//GENERAL
OP40_Auto:					BOOL;
OP40_HomeRunning:			BOOL;
OP40_ErrorActive:			BOOL;
OP40_Home_PB:				BOOL;
OP40_Work_PB:				BOOL;
OP40_ManualSafetyBypass:	BOOL;
OP40_LightCurtainBypass:	BOOL;
OP40_OperationCompleted:	BOOL;
OP40_LampCheck:				BOOL;
OP40_MachineLamp:			BOOL;
OP40_ComponentOk:			BOOL;
OP40_ComponentNok:			BOOL;
OP40_RepeatBit:				BOOL;
OP40_HomingResetBit:		BOOL;
OP40_ControlledByRobo:		BOOL;
OP40_Any_Bypass:			BOOL;
OP40_ManualModeStatus:		INT;
OP40_ManualModeWord:		INT;
OP40_AutoRunning:			BOOL;
OP40_StepRunning:			BOOL;
OP40_StartEnable:   		BOOL;
OP40_Machine_Stop: 			BOOL;
OP40_AutoSeq:				INT;
OP40_LH_AutoSeq: 			INT;
OP40_RH_AutoSeq: 			INT;
OP40_Homing_Seq:			INT;
OP40_HomeConditionOK:   	BOOL;
OP40_Safety_OK:				BOOL;
OP40_Mode_Ack:				BOOL;
OP40_Temp_hmeOK:			BOOL;
OP40_Stop_Request: BOOL;

//Automatic_Run:				BOOL;

OP40_Prev_Stat_Operation_Completed: BOOL;
OP40_Prev_Comp_Status: INT;
OP40_Prev_LH_COMP_OK:BOOL;
OP40_Prev_LH_COMP_NOK:BOOL;
OP40_Prev_RH_COMP_OK:BOOL;
OP40_Prev_RH_COMP_NOK:BOOL;
OP40_LH_Operation_Completed:BOOL;
OP40_RH_Operation_Completed:BOOL;

//ModeSelection Outputs
//OP130_AutoSelected:		    BOOL;
OP40_ManualSelected:		BOOL;
OP40_StepSelected:			BOOL;
OP40_AutoSelected:		    BOOL;


//HMI Tags(From HMI)
OP40_HMI_AutoMode:						BOOL;
OP40_HMI_ManualMOde:					BOOL;
OP40_HMI_StepMode:						BOOL;
OP40_HMI_CycleStart:					BOOL;
OP40_HMI_Cycle_Start:					BOOL;
OP40_HMI_Reset:						    BOOL;
OP40_HMI_Homing:						BOOL;
SR40_Vert_Servo_Max_Lim:				BOOL;



//Servo
SR40_Vert_servo : FB_Axis;
SR40_Vert_servo_ctrl:Servo_Control;
SR40_Vert_servo_not_Home: BOOL;
SR40_Vert_servo_status:stManualModeAxis;
SR40_Vert_servo_Axis :AXIS_REF;

//MANUAL	
	OP40_man_cyl_no 				: INT;
	
//AUTO	

	OP40_AUTO_STP_NO				: INT;


// SERVO VARIABLE
	OP40_VERT_SERVO_STRT			: BOOL;				// SERVO MOVE TO TARGET POSITION
	OP40_SERVO_POS_DONE				: BOOL;				// SERVO POSITION REACHED
	OP40_SERVO_ON_SFE_WRK			: BOOL;				// SERVO ACTUAL POSITION = SERVO SAFE POSITION
	OP40_SERVO_ON_WRK_1				: BOOL;				// SERVO ACTUAL POSITION = SERVO WORK POSITION
	OP40_SERVO_ON_WRK_2				: BOOL;	
    OP40_SERVO_ON_HOME				: BOOL;				// SERVO ACTUAL POSITION = SERVO HOME POSITION		  
	OP40_VERT_SERVO_POSITION		: REAL;				// SERVO ACTUAL POSITION

//LVDT

OP40_LH AT %I*:  DINT;
OP40_RH AT %I*:  DINT;
OP60_LH AT %I*:  DINT;
OP60_RH AT %I*:  DINT;
OP80_LH AT %I*:  DINT;
OP80_RH AT %I*:  DINT;



END_VAR

VAR_GLOBAL PERSISTENT
//LVDT 
	OP40_SET_LVDT_VALUE				:LREAL;	           // FROM HMI OR RECIPE
	OP40_LVDT_TOLERANCE 			:LREAL;			   // FROM HMI OR RECIPE
	OP40_LH_LVDT_VALUE				:REAL;			   // FROM LVDT
	OP40_RH_LVDT_VALUE				:REAL;
	
	OP40_Cycle_Time : UDINT;
//Error
	OP40_ErrorWord_0: DINT;
	OP40_ErrorWord_1: DINT;
	OP40_ErrorWord_2: DINT;	
// MANUAL
	OP40_STN_ENABLE					: BOOL;				// FROM MASTER CONTROL BLOCK 
	OP40_STN_RUNNING				: BOOL;
// AUTO
	OP40_BYPASS						: BOOL;				// OP40 ON-BYPASS
	OP40_LH_LVDT_OK					: BOOL;				// TO MASTER CONTROL BLOCK LH OK BIT
	OP40_LH_LVDT_NOK				: BOOL;				// TO MASTER CONTROL BLOCK LH NOK BIT
	OP40_RH_LVDT_OK					: BOOL;				// TO MASTER CONTROL BLOCK RH OK BIT
	OP40_RH_LVDT_NOK				: BOOL;				// TO MASTER CONTROL BLOCK RH NOK BIT		  
	OP40_DLY_AFT_SFE_WRK			: INT  := 200;		// AUTO DELAY TIMER AFTER SERVO REACH WORK
	
	OP40_HMI_LH_LVDT_VALUE				: REAL;
	OP40_HMI_RH_LVDT_VALUE				: REAL;

//SERVO	
	OP40_VERT_SERVO_HME_POS			: REAL :=0;             // SERVO HOME POSITION FROM HMI
	OP40_VERT_SERVO_SFE_WRK_POS		: REAL :=0;				// SERVO SAFE WORK POSITION FROM RECEIPE
	OP40_VERT_SERVO_WRK_POS_1		: REAL :=35;
    OP40_VERT_SERVO_WRK_POS_2		: REAL :=40;		// SERVO WORK POSITION FROM RECEIPE	
	OP40_VERT_SERVO_TARGET			: REAL;				// SERVO AUTO TARGET POSITION	

//Setting Parameters
    OP40_HMI_Servo_Speed   : REAL;
    OP40_HMI_Servo_Speed_Offset : REAL;
	OP40_HMI_Servo_Pos_Offset   : REAL;	
    OP40_HMI_Low_Limit		 : REAL;
    OP40_HMI_High_Limit		 : REAL;
	OP40_HMI_Safe_Home		 : REAL;
	OP40_HMI_Safe_Work		 : REAL;
END_VAR

// ---- POUs/Programs/OP40/OP40_Recipe.TcGVL

VAR_GLOBAL PERSISTENT
	OP40_DLY_BEF_MEAS : INT;
	OP40_VERT_SERVO_WORK_POS : REAL;
	OP40_VERT_SERVO_SFE_WORK_POS : REAL;	
END_VAR

// ---- POUs/Programs/OP50/OP50_GVL.TcGVL
VAR_GLOBAL
			
//GENERAL
OP50_Auto:					BOOL;
OP50_Mode_Ack:				BOOL;
OP50_HomeRunning:			BOOL;
OP50_ErrorActive:			BOOL;
OP50_Home_PB:				BOOL;
OP50_Work_PB:				BOOL;
OP50_ManualSafetyBypass:	BOOL;
OP50_LightCurtainBypass:	BOOL;
OP50_OperationCompleted:	BOOL;
OP50_LampCheck:				BOOL;
OP50_MachineLamp:			BOOL;
OP50_ComponentOk:			BOOL;
OP50_ComponentNok:			BOOL;
OP50_RepeatBit:				BOOL;
OP50_HomingResetBit:		BOOL;
OP50_ControlledByRobo:		BOOL;
OP50_Any_Bypass:			BOOL;
OP50_ManualModeStatus:		INT;
OP50_ManualModeWord:		INT;
OP50_AutoRunning:			BOOL;
OP50_StepRunning:			BOOL;
OP50_StartEnable:   		BOOL;
OP50_HomeConditionOK:		BOOL;
OP50_Temp_hmeOK:			BOOL;
OP50_Machine_Stop: 			BOOL;
OP50_AutoSeq:				INT;
OP50_LH_AutoSeq: 			INT;
OP50_RH_AutoSeq: 			INT;
OP50_Homing_Seq:			INT;
OP50_Safety_OK:				BOOL;
OP50_STN_ENABLE				: BOOL;
OP50_Stop_Request: BOOL;	
OP50_Conveyor_Run			: BOOL;
	
OP50_ManualSelected:		BOOL;
OP50_StepSelected:			BOOL;
OP50_AutoSelected:		    BOOL;

OP50_HMI_AutoMode:						BOOL;
OP50_HMI_ManualMode:					BOOL;
OP50_HMI_StepMode:						BOOL;
OP50_HMI_CycleStart:					BOOL;
OP50_HMI_Cycle_Start:					BOOL;

OP50_HMI_Homing:						BOOL;

SR50_Vert_servo: FB_Axis;
SR50_Hori_servo: FB_Axis;
SR50_Conv_servo: FB_Axis;
OP50_GIUDE_GRP: FB_Axis_FESTO;

Drum_feeder_ON 	  : BOOL;
Drum_feeder_State : BOOL;

Camera_LH_Trig : BOOL;
Camera_LH_OK   : BOOL;

Camera_RH_Trig : BOOL;
Camera_RH_OK   : BOOL;

//Cylinder
CR50_LH_Rej_Cyl: Cylinder_Block;
CR50_RH_Rej_Cyl: Cylinder_Block;
CR50_LH_Grip_Cyl: Cylinder_Block;
CR50_RH_Grip_Cyl: Cylinder_Block;
CR50_LH_Rej_Cyl_status : INT;
CR50_RH_Rej_Cyl_status : INT;
CR50_LH_Grip_Cyl_status : INT;
CR50_RH_Grip_Cyl_status : INT;
OP50_HMI_LH_Rej_Cyl_Home_PB : BOOL;
OP50_HMI_LH_Rej_Cyl_Work_PB : BOOL;
OP50_HMI_RH_Rej_Cyl_Home_PB : BOOL;
OP50_HMI_RH_Rej_Cyl_Work_PB : BOOL;
OP50_HMI_LH_Grip_Cyl_Home_PB : BOOL;
OP50_HMI_LH_Grip_Cyl_Work_PB : BOOL;
OP50_HMI_RH_Grip_Cyl_Home_PB : BOOL;
OP50_HMI_RH_Grip_Cyl_Work_PB : BOOL;
//conveyor
OP50_pick_ready     : BOOL;
OP50_pick_done      : BOOL;
OP50_Conv_Fwd_Time	: INT;
OP50_Conv_Rev_Time	: INT;
OP50_Conveyor_FWD_Speed	: REAL;
OP50_Conveyor_REV_Speed	: REAL;
// Sensors

	
//Camera GVLs
	OP50_Camera_Trigger				  : BOOL;
	OP50_LH_Clr_OK					  : BOOL;
	OP50_LH_Clr_NOK					  : BOOL;
	OP50_LH_Size_OK					  : BOOL;
	OP50_LH_Size_NOK				  : BOOL;
	OP50_LH_Part_OK					  : BOOL;
	OP50_LH_Part_NOK				  : BOOL;
	
	OP50_Size_Rej					  : BOOL;
	OP50_Size_Rej_Complete			  : BOOL;
	OP50_One_Cycle				      : BOOL;
	OP50_LH_Camera_OK 				  : BOOL;
	OP50_LH_Camera_NOK                : BOOL;
	OP50_RH_Camera_OK                 : BOOL;
	OP50_RH_Camera_NOK                : BOOL;
	OP50_Camera_Done				  : BOOL;
	
	OP50_RH_Clr_OK					  : BOOL;
	OP50_RH_Clr_NOK					  : BOOL;
	OP50_RH_Size_OK					  : BOOL;
	OP50_RH_Size_NOK				  : BOOL;
	OP50_RH_Part_OK					  : BOOL;
	OP50_RH_Part_NOK				  : BOOL;
	
	OP50_LH_Camera_Trigger		      : BOOL;
	OP50_LH_Camera_Job_Change_start   : BOOL;
	OP50_LH_Camera_Error			  : BOOL;
	OP50_LH_Camera_Ready			  : BOOL;
	OP50_LH_Camera_Online			  : BOOL;	
	OP50_LH_Job_Change_Complete		    : BOOL;
	OP50_LH_Job_Change_Error   		    : BOOL;
	OP50_LH_Picture_Taken      		    : BOOL;	
	OP50_LH_Error_status			    : STRING;
	OP50_LH_Target_Job_ID				: UINT;
	OP50_LH_Loaded_Job_ID		    	: UINT;
	
	OP50_RH_Camera_Trigger		      : BOOL;
	OP50_RH_Camera_Job_Change_start   : BOOL;
	OP50_RH_Camera_Error			  : BOOL;
	OP50_RH_Camera_Ready			  : BOOL;
	OP50_RH_Camera_Online			  : BOOL;
	OP50_RH_Job_Change_Complete		    : BOOL;
	OP50_RH_Job_Change_Error   		    : BOOL;
	OP50_RH_Picture_Taken      		    : BOOL;
	OP50_RH_Error_status				: STRING;
	OP50_RH_Target_Job_ID				: UINT;
	OP50_RH_Loaded_Job_ID		    	: UINT;		
	
END_VAR

VAR_GLOBAL PERSISTENT
	OP50_Gripper_LH_Open  : BOOL;
    OP50_Gripper_LH_Close : BOOL;
    OP50_Gripper_LH_State : BOOL;  //1-- Open 0--Close
    
    OP50_Gripper_RH_Open  : BOOL;
    OP50_Gripper_RH_Close : BOOL;
    OP50_Gripper_RH_State : BOOL;


    OP50_VERT_SERVO_POS_DONE	    	: BOOL;
    OP50_VERT_SERVO_ON_SFE_WRK			: BOOL;
    OP50_VERT_SERVO_ON_WRK_PICK			: BOOL;
	OP50_VERT_SERVO_ON_WRK_PLACE		: BOOL;
    OP50_VERT_SERVO_ON_HOME				: BOOL;
	  
	OP50_VERT_SERVO_POSITION		: LREAL ;
	OP50_VERT_SERVO_HME_POS			: REAL := 0;  				
	OP50_VERT_SERVO_SFE_WRK_POS		: REAL :=10;		
	OP50_VERT_SERVO_PICK_POS		: REAL :=58.5;	
	OP50_VERT_SERVO_PLACE_POS		: REAL :=40;

	OP50_Conv_Fwd_Pos				: REAL :=10;
	OP50_Conv_Rev_Pos				: REAL :=5;	
	
    OP50_HORI_SERVO_POS_DONE	    	: BOOL;
    OP50_HORI_SERVO_ON_SFE_WRK			: BOOL;
    OP50_HORI_SERVO_ON_WRK_PICK			: BOOL;
    OP50_HORI_SERVO_ON_SFE_WRK_PICK		: BOOL;		
	OP50_HORI_SERVO_ON_WRK_PLACE		: BOOL;
    OP50_HORI_SERVO_ON_HOME				: BOOL;
	  
	OP50_HORI_SERVO_POSITION		: LREAL ;
	OP50_HORI_SERVO_HME_POS			: REAL :=-40;  				
	OP50_HORI_SERVO_SFE_WRK_POS		: REAL :=-40;
	OP50_HORI_SERVO_SAFE_PICK_POS	: REAL := 110; 		
	OP50_HORI_SERVO_PICK_POS		: REAL :=151;	
	OP50_HORI_SERVO_PLACE_POS		: REAL :=74;
	
    OP50_CONV_SERVO_POS_DONE	    	: BOOL;
    OP50_CONV_SERVO_ON_SFE_WRK			: BOOL;
    OP50_CONV_SERVO_ON_WRK				: BOOL;
    OP50_CONV_SERVO_ON_HOME				: BOOL;
	
	OP50_CONV_SERVO_POSITION		: LREAL ;
	OP50_CONV_SERVO_HME_POS			: REAL;  				
	OP50_CONV_SERVO_SFE_WRK_POS		: REAL ;		
	OP50_CONV_SERVO_WRK_POS			: REAL;

//Error
OP50_ErrorWord_0: DINT;
OP50_ErrorWord_1: DINT;
OP50_ErrorWord_2: DINT;	

	OP50_Cycle_Time : UDINT;

//Drum_Feeder
	OP50_Drum_Feed_Motor_Speed		AT %Q*  : INT;	
	OP50_HMI_Drum_Feed_Mtr_Speed_IP		: INT;
	OP50_Drum_Feed_Mtr_Speed_Select		: BOOL;
	OP50_Drum_Feed_Mtr_Run_Fwd 			: BOOL;
	OP50_Drum_Feed_Mtr_Reset   			: BOOL;

//Setting Parameters
    OP50_HMI_Servo_Speed_Vertical     : REAL ;
	OP50_HMI_Servo_Speed_Horizontal	  : REAL ;
    OP50_HMI_Hori_Low_Limit		 : REAL:=0;
    OP50_HMI_Hori_High_Limit     : REAL:=200;
    OP50_HMI_Vert_Low_Limit		 : REAL:=0;
    OP50_HMI_Vert_High_Limit     : REAL:=100;	

	OP50_Vert_Ser_Safe_Pos			: REAL;
	OP50_Hori_Ser_Rej_Pos			: REAL;	
	OP50_Hori_Ser_Jerk_Pos			: REAL :=2;		
	OP50_Drum_Freq		  			: REAL;
	
	OP50_Conv_Fwd_Time_6_3			: INT:=750;
	OP50_Conv_Fwd_Speed_6_3			: INT:=150;
	OP50_Conv_Rev_Time_6_3			: INT:=500;
	OP50_Conv_Rev_Speed_6_3			: INT:=-100;

	OP50_Conv_Fwd_Time_7_89			: INT:=750;
	OP50_Conv_Fwd_Speed_7_89		: INT:=150;
	OP50_Conv_Rev_Time_7_89			: INT:=500;
	OP50_Conv_Rev_Speed_7_89		: INT:=-100;		
	
	OP50_Conveyor_Speed				: REAL;
	OP50_Model						: STRING[80];

	OP50_Grip_LH_Bypass				: BOOL;
	OP50_Grip_RH_Bypass				: BOOL;	
	OP50_Guide_Pos					: REAL :=75;
//Drum Timers
	OP50_Drum_ON_Time				: INT:=4000;
	OP50_Drum_OFF_Time				: INT:=1000;
	
	
END_VAR

// ---- POUs/Programs/OP50/OP50_HMI_GVL.TcGVL

VAR_GLOBAL
	
OP50_HMI_Reset:						    BOOL;
SR50_Vert_servo_ctrl:Servo_Control;
SR50_Vert_servo_status:stManualModeAxis;

SR50_Hori_servo_ctrl:Servo_Control;
SR50_Hori_servo_status:stManualModeAxis;


SR50_Conv_servo_ctrl:Servo_Control;
SR50_Conv_servo_status:stManualModeAxis;


OP50_GIUDE_GRP_Manual_Axis: stManualModeAxis; 
OP50_GIUDE_GRP_ctrl: Servo_Control;
END_VAR

// ---- POUs/Programs/OP50/OP50_Recipe.TcGVL

VAR_GLOBAL
END_VAR

// ---- POUs/Programs/OP60/OP60_GVL.TcGVL
VAR_GLOBAL
	
//GENERAL
OP60_Auto:					BOOL;
OP60_HomeRunning:			BOOL;
OP60_ErrorActive:			BOOL;
OP60_Home_PB:				BOOL;
OP60_Work_PB:				BOOL;
OP60_ManualSafetyBypass:	BOOL;
OP60_LightCurtainBypass:	BOOL;
OP60_OperationCompleted:	BOOL;
OP60_LampCheck:				BOOL;
OP60_MachineLamp:			BOOL;
OP60_ComponentOk:			BOOL;
OP60_ComponentNok:			BOOL;
OP60_RepeatBit:				BOOL;
OP60_HomingResetBit:		BOOL;
OP60_ControlledByRobo:		BOOL;
OP60_Any_Bypass:			BOOL;
OP60_ManualModeStatus:		INT;
OP60_ManualModeWord:		INT;
OP60_AutoRunning:			BOOL;
OP60_StepRunning:			BOOL;
OP60_StartEnable:   		BOOL;
OP60_Machine_Stop: 			BOOL;
OP60_AutoSeq:				INT;
OP60_LH_AutoSeq: 			INT;
OP60_RH_AutoSeq: 			INT;
OP60_Homing_Seq:			INT;
OP60_HomeConditionOK:   	BOOL;
OP60_Safety_OK:				BOOL;
OP60_Mode_Ack:				BOOL;
OP60_Temp_hmeOK:			BOOL;
OP60_Stop_Request: BOOL;

Automatic_Run:				BOOL;

OP60_Prev_Stat_Operation_Completed: BOOL;
OP60_Prev_Comp_Status: INT;
OP60_Prev_LH_COMP_OK:BOOL;
OP60_Prev_LH_COMP_NOK:BOOL;
OP60_Prev_RH_COMP_OK:BOOL;
OP60_Prev_RH_COMP_NOK:BOOL;
OP60_LH_Operation_Completed:BOOL;
OP60_RH_Operation_Completed:BOOL;

//ModeSelection Outputs
//OP130_AutoSelected:		    BOOL;
OP60_ManualSelected:		BOOL;
OP60_StepSelected:			BOOL;
OP60_AutoSelected:		    BOOL;


//HMI Tags(From HMI)
OP60_HMI_AutoMode:						BOOL;
OP60_HMI_ManualMOde:					BOOL;
OP60_HMI_StepMode:						BOOL;
OP60_HMI_CycleStart:					BOOL;
OP60_HMI_Cycle_Start:					BOOL;
OP60_HMI_Reset:						    BOOL;
OP60_HMI_Homing:						BOOL;
SR60_Vert_Servo_Max_Lim:				BOOL;



//Servo
SR60_Vert_servo : FB_Axis;
SR60_Vert_servo_ctrl:Servo_Control;
SR60_Vert_servo_not_Home: BOOL;
SR60_Vert_servo_status:stManualModeAxis;
SR60_Vert_servo_Axis :AXIS_REF;

//MANUAL	
	OP60_man_cyl_no 				: INT;
	
//AUTO	

	OP60_AUTO_STP_NO				: INT;


// SERVO VARIABLE
	OP60_VERT_SERVO_STRT			: BOOL;				// SERVO MOVE TO TARGET POSITION
	OP60_SERVO_POS_DONE				: BOOL;				// SERVO POSITION REACHED
// SERVO ACTUAL POSITION
	
END_VAR

VAR_GLOBAL PERSISTENT
//LVDT 
	OP60_SET_LVDT_VALUE				:LREAL;	           // FROM HMI OR RECIPE
	OP60_LVDT_TOLERANCE 			:LREAL;			   // FROM HMI OR RECIPE
	OP60_LH_LVDT_VALUE				:LREAL;			   // FROM LVDT
	OP60_RH_LVDT_VALUE				:LREAL;
	
// MANUAL
	OP60_Cycle_Time : UDINT;
// AUTO
	OP60_BYPASS						: BOOL;				// OP60 ON-BYPASS
	OP60_LH_LVDT_OK					: BOOL;				// TO MASTER CONTROL BLOCK LH OK BIT
	OP60_LH_LVDT_NOK				: BOOL;				// TO MASTER CONTROL BLOCK LH NOK BIT
	OP60_RH_LVDT_OK					: BOOL;				// TO MASTER CONTROL BLOCK RH OK BIT
	OP60_RH_LVDT_NOK				: BOOL;				// TO MASTER CONTROL BLOCK RH NOK BIT

	OP60_HMI_LH_LVDT_VALUE				: REAL;
	OP60_HMI_RH_LVDT_VALUE				: REAL;	
	  
	OP60_DLY_AFT_SFE_WRK			: INT := 200;				// AUTO DELAY TIMER AFTER SERVO REACH WORK

//SERVO	
	OP60_SERVO_ON_WRK_1				: BOOL;				// SERVO ACTUAL POSITION = SERVO WORK POSITION
	OP60_SERVO_ON_WRK_2				: BOOL;	
	OP60_SERVO_ON_SFE_WRK			: BOOL;				// SERVO ACTUAL POSITION = SERVO SAFE POSITION
	OP60_SERVO_ON_HOME				: BOOL;				// SERVO ACTUAL POSITION = SERVO HOME POSITION
	OP60_VERT_SERVO_POSITION		: REAL;					
    OP60_VERT_SERVO_SFE_WRK_POS		: REAL;
	OP60_VERT_SERVO_HME_POS			: REAL;
	OP60_VERT_SERVO_WRK_POS_1       : REAL;
	OP60_VERT_SERVO_WRK_POS_2       : REAL;
//Setting Parameters
    OP60_HMI_Servo_Speed        : REAL;
    OP60_HMI_Servo_Speed_Offset : REAL;
	OP60_HMI_Servo_Pos_Offset   : REAL;		
    OP60_HMI_Low_Limit		 : REAL;
    OP60_HMI_High_Limit		 : REAL;
	OP60_HMI_Safe_Home		 : REAL;
	OP60_HMI_Safe_Work		 : REAL;

	OP60_STN_ENABLE			 : BOOL;				// FROM MASTER CONTROL BLOCK 
	OP60_STN_RUNNING    	 : BOOL;	
//Error
	OP60_ErrorWord_0: DINT;
	OP60_ErrorWord_1: DINT;
	OP60_ErrorWord_2: DINT;	
END_VAR

// ---- POUs/Programs/OP60/OP60_Recipe.TcGVL
//{attribute 'qualified_only'}
VAR_GLOBAL PERSISTENT
	OP60_DLY_BEF_MEAS : INT;
	OP60_VERT_SERVO_WORK_POS : REAL;
	OP60_VERT_SERVO_SFE_WORK_POS : REAL;	
END_VAR

// ---- POUs/Programs/OP70/OP70_GVL.TcGVL

VAR_GLOBAL
			
//GENERAL
OP70_Auto:					BOOL;
OP70_Mode_Ack:				BOOL;
OP70_HomeRunning:			BOOL;
OP70_ErrorActive:			BOOL;
OP70_Home_PB:				BOOL;
OP70_Work_PB:				BOOL;
OP70_ManualSafetyBypass:	BOOL;
OP70_LightCurtainBypass:	BOOL;
OP70_OperationCompleted:	BOOL;
OP70_LampCheck:				BOOL;
OP70_MachineLamp:			BOOL;
OP70_ComponentOk:			BOOL;
OP70_ComponentNok:			BOOL;
OP70_RepeatBit:				BOOL;
OP70_HomingResetBit:		BOOL;
OP70_ControlledByRobo:		BOOL;
OP70_Any_Bypass:			BOOL;
OP70_ManualModeStatus:		INT;
OP70_ManualModeWord:		INT;
OP70_AutoRunning:			BOOL;
OP70_StepRunning:			BOOL;
OP70_StartEnable:   		BOOL;
OP70_HomeConditionOK:		BOOL;
OP70_Temp_hmeOK:			BOOL;
OP70_Machine_Stop: 			BOOL;
OP70_AutoSeq:				INT;
OP70_LH_AutoSeq: 			INT;
OP70_RH_AutoSeq: 			INT;
OP70_Homing_Seq:			INT;
OP70_Safety_OK:				BOOL;
OP70_STN_ENABLE				: BOOL;
OP70_Stop_Request			: BOOL;
OP70_Conveyor_ON			: BOOL;

OP70_ManualSelected:		BOOL;
OP70_StepSelected:			BOOL;
OP70_AutoSelected:		    BOOL;

OP70_HMI_AutoMode:						BOOL;
OP70_HMI_ManualMode:					BOOL;
OP70_HMI_StepMode:						BOOL;
OP70_HMI_CycleStart:					BOOL;
OP70_HMI_Cycle_Start:					BOOL;
OP70_HMI_Reset:						    BOOL;
OP70_HMI_Homing:						BOOL;

SR70_Vert_servo: FB_Axis;
SR70_Vert_servo_ctrl:Servo_Control;
SR70_Vert_servo_status:stManualModeAxis;

SR70_Hori_servo: FB_Axis;
SR70_Hori_servo_ctrl:Servo_Control;
SR70_Hori_servo_status:stManualModeAxis;

SR70_Conv_servo: FB_Axis;
SR70_Conv_servo_ctrl:Servo_Control;
SR70_Conv_servo_status:stManualModeAxis;

(*OP70_GIUDE_GRP: FB_Axis;*)
OP70_GUIDE_GRP	: FB_Axis_FESTO;
OP70_GIUDE_GRP_Manual_Axis: stManualModeAxis; 
OP70_GIUDE_GRP_ctrl: Servo_Control;



Drum_feeder_ON 	  : BOOL;
Drum_feeder_State : BOOL;

Camera_LH_Trig : BOOL;
Camera_LH_OK   : BOOL;

Camera_RH_Trig : BOOL;
Camera_RH_OK   : BOOL;

//Cylinder
CR70_LH_Rej_Cyl: Cylinder_Block;
CR70_RH_Rej_Cyl: Cylinder_Block;
CR70_LH_Rej_Cyl_status : INT;
CR70_RH_Rej_Cyl_status : INT;
OP70_HMI_LH_Rej_Cyl_Home_PB : BOOL;
OP70_HMI_LH_Rej_Cyl_Work_PB : BOOL;
OP70_HMI_RH_Rej_Cyl_Home_PB : BOOL;
OP70_HMI_RH_Rej_Cyl_Work_PB : BOOL;

//conveyor
OP70_pick_ready: BOOL;
OP70_pick_done : BOOL;
OP70_Conv_Fwd_Time	: INT;
OP70_Conv_Rev_Time	: INT;
OP70_Conveyor_FWD_Speed	: REAL;
OP70_Conveyor_REV_Speed	: REAL;
//Schunk
OP70_Gripper_LH : FB_Schunk;
OP70_Gripper_LH_Manual_Axis: stManualModeAxis; 
OP70_Gripper_LH_Gripper_ctrl: Servo_Control; 
  
OP70_Gripper_Current     : REAL;
OP70_Gripper_Acceleration: REAL;
OP70_Gripper_Jerk        : REAL;

OP70_Gripper_RH : FB_Schunk;
OP70_Gripper_RH_Manual_Axis: stManualModeAxis;
OP70_Gripper_RH_Gripper_ctrl: Servo_Control; 

	OP70_Camera_Done: BOOL;
	OP70_One_Cycle : BOOL;

//Camera GVLS
	OP70_LH_Camera_Trigger		      : BOOL;
	OP70_LH_Camera_Job_Change_start   : BOOL;
	OP70_LH_Camera_Error			  : BOOL;
	OP70_LH_Camera_Ready			  : BOOL;
	OP70_LH_Camera_Online			  : BOOL;	
	OP70_LH_Job_Change_Complete		    : BOOL;
	OP70_LH_Job_Change_Error   		    : BOOL;
	OP70_LH_Picture_Taken      		    : BOOL;
	OP70_LH_Error_status				: STRING;
	OP70_LH_Target_Job_ID				: UINT;
	OP70_LH_Loaded_Job_ID		    	: UINT;	

	OP70_RH_Camera_Trigger		      : BOOL;
	OP70_RH_Camera_Job_Change_start   : BOOL;
	OP70_RH_Camera_Error			  : BOOL;
	OP70_RH_Camera_Ready			  : BOOL;
	OP70_RH_Camera_Online			  : BOOL;	
	OP70_RH_Job_Change_Complete		    : BOOL;
	OP70_RH_Job_Change_Error   		    : BOOL;
	OP70_RH_Picture_Taken      		    : BOOL;
	OP70_RH_Error_status				: STRING;
	OP70_RH_Target_Job_ID				: UINT;
	OP70_RH_Loaded_Job_ID		    	: UINT;	
	
END_VAR

VAR_GLOBAL PERSISTENT
	
	OP70_Conv_Fwd_Pos				: REAL :=10;
	OP70_Conv_Rev_Pos				: REAL  :=5;

	OP70_Gripper_Wrk_POS  : LREAL	:=2;
	OP70_Gripper_LH_Open  : BOOL;
    OP70_Gripper_LH_Close : BOOL;
    OP70_Gripper_LH_State : BOOL;  //1-- Open 0--Close
 
    OP70_Gripper_RH_Open  : BOOL;
    OP70_Gripper_RH_Close : BOOL;
    OP70_Gripper_RH_State : BOOL;

    OP70_VERT_SERVO_POS_DONE	    	: BOOL;
    OP70_VERT_SERVO_ON_SFE_WRK			: BOOL;
    OP70_VERT_SERVO_ON_WRK_PICK			: BOOL;
	OP70_VERT_SERVO_ON_WRK_PLACE		: BOOL;
    OP70_VERT_SERVO_ON_HOME				: BOOL;
	  
	OP70_VERT_SERVO_POSITION		: LREAL ;
	OP70_VERT_SERVO_HME_POS			: REAL := 0;  				
	OP70_VERT_SERVO_SFE_WRK_POS		: REAL :=10;		
	OP70_VERT_SERVO_PICK_POS		: REAL ;	
	OP70_VERT_SERVO_PLACE_POS		: REAL ;

    OP70_HORI_SERVO_POS_DONE	    	: BOOL;
    OP70_HORI_SERVO_ON_SFE_WRK			: BOOL;
    OP70_HORI_SERVO_ON_WRK_PICK			: BOOL;
    OP70_HORI_SERVO_ON_SFE_WRK_PICK		: BOOL;	
	OP70_HORI_SERVO_ON_WRK_PLACE		: BOOL;
    OP70_HORI_SERVO_ON_HOME				: BOOL;
	  
	OP70_HORI_SERVO_POSITION		: LREAL ;
	OP70_HORI_SERVO_HME_POS			: REAL := -40;  				
	OP70_HORI_SERVO_SFE_WRK_POS		: REAL := -40;
	OP70_HORI_SERVO_SAFE_PICK_POS	: REAL := 100; 		
	OP70_HORI_SERVO_PICK_POS		: REAL ;	
	OP70_HORI_SERVO_PLACE_POS		: REAL ;
	
    OP70_CONV_SERVO_POS_DONE	    	: BOOL;
    OP70_CONV_SERVO_ON_SFE_WRK			: BOOL;
    OP70_CONV_SERVO_ON_WRK				: BOOL;
    OP70_CONV_SERVO_ON_HOME				: BOOL;
	
	OP70_CONV_SERVO_POSITION		: LREAL ;
	OP70_CONV_SERVO_HME_POS			: REAL;// := 0;  				
	OP70_CONV_SERVO_SFE_WRK_POS		: REAL ;//:= 40;		
	OP70_CONV_SERVO_WRK_POS			: REAL;// := 200;	

//Error
OP70_ErrorWord_0: DINT;
OP70_ErrorWord_1: DINT;
OP70_ErrorWord_2: DINT;

	OP70_Cycle_Time : UDINT;

//Drum_Feeder
	OP70_Drum_Feed_Motor_Speed		AT %Q*  : INT;	
	OP70_HMI_Drum_Feed_Mtr_Speed_IP		: INT;
	OP70_Drum_Feed_Mtr_Speed_Select		: BOOL;
	OP70_Drum_Feed_Mtr_Run_Fwd 			: BOOL;
	OP70_Drum_Feed_Mtr_Reset   			: BOOL;	

//Setting Parameters

    OP70_HMI_Servo_Speed_Vertical     : REAL ;
	OP70_HMI_Servo_Speed_Horizontal	  : REAL ;
    OP70_HMI_Hori_Low_Limit		 : REAL;
    OP70_HMI_Hori_High_Limit     : REAL;
    OP70_HMI_Vert_Low_Limit		 : REAL;
    OP70_HMI_Vert_High_Limit     : REAL;	

	OP70_Vert_Ser_Safe_Pos			: REAL;
	OP70_Hori_Ser_Rej_Pos			: REAL;	
	OP70_Hori_Ser_Jerk_Pos			: REAL :=1;		
	OP70_Drum_Freq		  			: REAL;
	
	OP70_Conv_Fwd_Time_6_3			: INT:=750;
	OP70_Conv_Fwd_Speed_6_3			: INT:=150;
	OP70_Conv_Rev_Time_6_3			: INT:=500;
	OP70_Conv_Rev_Speed_6_3			: INT:=-100;

	OP70_Conv_Fwd_Time_7_89			: INT:=750;
	OP70_Conv_Fwd_Speed_7_89		: INT:=150;
	OP70_Conv_Rev_Time_7_89			: INT:=500;
	OP70_Conv_Rev_Speed_7_89		: INT:=-100;	
	
	OP70_Model: STRING[80];
	OP70_Conveyor_Speed				: REAL;
	OP70_Grip_LH_Bypass				: BOOL;
	OP70_Grip_RH_Bypass				: BOOL;
	OP70_Guide_Pos					: REAL :=70;	
	
//Drum Timers
	OP70_Drum_ON_Time				: INT:=4000;
	OP70_Drum_OFF_Time				: INT:=1000;		
END_VAR

// ---- POUs/Programs/OP70/OP70_Recipe.TcGVL

VAR_GLOBAL
END_VAR

// ---- POUs/Programs/OP80/OP80_GVL.TcGVL
VAR_GLOBAL
	
//GENERAL
OP80_Auto:					BOOL;
OP80_HomeRunning:			BOOL;
OP80_ErrorActive:			BOOL;
OP80_Home_PB:				BOOL;
OP80_Work_PB:				BOOL;
OP80_ManualSafetyBypass:	BOOL;
OP80_LightCurtainBypass:	BOOL;
OP80_OperationCompleted:	BOOL;
OP80_LampCheck:				BOOL;
OP80_MachineLamp:			BOOL;
OP80_ComponentOk:			BOOL;
OP80_ComponentNok:			BOOL;
OP80_RepeatBit:				BOOL;
OP80_HomingResetBit:		BOOL;
OP80_ControlledByRobo:		BOOL;
OP80_Any_Bypass:			BOOL;
OP80_ManualModeStatus:		INT;
OP80_ManualModeWord:		INT;
OP80_AutoRunning:			BOOL;
OP80_StepRunning:			BOOL;
OP80_StartEnable:   		BOOL;
OP80_Machine_Stop: 			BOOL;
OP80_AutoSeq:				INT;
OP80_LH_AutoSeq: 			INT;
OP80_RH_AutoSeq: 			INT;
OP80_Homing_Seq:			INT;
OP80_HomeConditionOK:   	BOOL;
OP80_Safety_OK:				BOOL;
OP80_Mode_Ack:				BOOL;
OP80_Temp_hmeOK:			BOOL;
OP80_Stop_Request: BOOL;

//Automatic_Run:				BOOL;

OP80_Prev_Stat_Operation_Completed: BOOL;
OP80_Prev_Comp_Status: INT;
OP80_Prev_LH_COMP_OK:BOOL;
OP80_Prev_LH_COMP_NOK:BOOL;
OP80_Prev_RH_COMP_OK:BOOL;
OP80_Prev_RH_COMP_NOK:BOOL;
OP80_LH_Operation_Completed:BOOL;
OP80_RH_Operation_Completed:BOOL;

//ModeSelection Outputs
//OP130_AutoSelected:		    BOOL;
OP80_ManualSelected:		BOOL;
OP80_StepSelected:			BOOL;
OP80_AutoSelected:		    BOOL;


//HMI Tags(From HMI)
OP80_HMI_AutoMode:						BOOL;
OP80_HMI_ManualMOde:					BOOL;
OP80_HMI_StepMode:						BOOL;
OP80_HMI_CycleStart:					BOOL;
OP80_HMI_Cycle_Start:					BOOL;
OP80_HMI_Reset:						    BOOL;
OP80_HMI_Homing:						BOOL;
SR80_Vert_Servo_Max_Lim:				BOOL;

//Servo
SR80_Vert_servo : FB_Axis;

SR80_Vert_servo_not_Home: BOOL;

//MANUAL	
	OP80_man_cyl_no 				: INT;
	
//AUTO	
	OP80_AUTO_STP_NO				: INT;


// SERVO VARIABLE
	OP80_VERT_SERVO_POSITION		: REAL;				// SERVO ACTUAL POSITION
	
END_VAR

VAR_GLOBAL PERSISTENT
//LVDT 
	OP80_SET_LVDT_VALUE				:LREAL;	           // FROM HMI OR RECIPE
	OP80_LVDT_TOLERANCE 			:LREAL;			   // FROM HMI OR RECIPE
	OP80_LH_LVDT_VALUE				:LREAL;			   // FROM LVDT
	OP80_RH_LVDT_VALUE				:LREAL;	
// MANUAL

// AUTO
	OP80_BYPASS						: BOOL;				// OP80 ON-BYPASS
	OP80_LH_LVDT_OK					: BOOL;				// TO MASTER CONTROL BLOCK LH OK BIT
	OP80_LH_LVDT_NOK				: BOOL;				// TO MASTER CONTROL BLOCK LH NOK BIT
	OP80_RH_LVDT_OK					: BOOL;				// TO MASTER CONTROL BLOCK RH OK BIT
	OP80_RH_LVDT_NOK				: BOOL;				// TO MASTER CONTROL BLOCK RH NOK BIT	
	  
	OP80_DLY_AFT_SFE_WRK			: INT := 200;				// AUTO DELAY TIMER AFTER SERVO REACH WORK

//SERVO	
	OP80_VERT_SERVO_HME_POS			: REAL ;             // SERVO HOME POSITION FROM HMI
	OP80_VERT_SERVO_SFE_WRK_POS		: REAL ;				// SERVO SAFE WORK POSITION FROM RECEIPE
	OP80_VERT_SERVO_WRK_POS			: REAL ;				// SERVO WORK POSITION FROM RECEIPE	
	OP80_VERT_SERVO_TARGET			: REAL;				// SERVO AUTO TARGET POSITION	

	OP80_SERVO_ON_WRK_1				: BOOL;	
	OP80_SERVO_ON_WRK_2				: BOOL;	
	OP80_SERVO_ON_SFE_WRK			: BOOL;	
	OP80_SERVO_ON_HOME				: BOOL;	
	//OP80_VERT_SERVO_POSITION		: REAL;	
    //OP80_VERT_SERVO_SFE_WRK_POS		: REAL;	
	//OP80_VERT_SERVO_HME_POS			: REAL;	
	OP80_VERT_SERVO_WRK_POS_1       : REAL;	
	OP80_VERT_SERVO_WRK_POS_2       : REAL;	
	OP80_HMI_LH_LVDT_VALUE				: REAL;
	OP80_HMI_RH_LVDT_VALUE				: REAL;		
	
	
	
//Setting Parameters
    OP80_HMI_Servo_Speed     : REAL;
    OP80_HMI_Servo_Speed_Offset : REAL;
	OP80_HMI_Servo_Pos_Offset   : REAL;	
    OP80_HMI_Low_Limit		 : REAL;
    OP80_HMI_High_Limit		 : REAL;
	OP80_HMI_Safe_Home		 : REAL;
	OP80_HMI_Safe_Work		 : REAL;
      
	OP80_STN_ENABLE			 : BOOL;				// FROM MASTER CONTROL BLOCK 
	OP80_STN_RUNNING 	     : BOOL;
//Error
	OP80_ErrorWord_0: DINT;
	OP80_ErrorWord_1: DINT;
	OP80_ErrorWord_2: DINT;		
	
	OP80_Cycle_Time : UDINT;
	
END_VAR

// ---- POUs/Programs/OP80/OP80_HMI_GVL.TcGVL

VAR_GLOBAL
	
SR80_Vert_servo_status:stManualModeAxis;
SR80_Vert_servo_ctrl:Servo_Control;
END_VAR

// ---- POUs/Programs/OP80/OP80_Recipe.TcGVL
//{attribute 'qualified_only'}
VAR_GLOBAL PERSISTENT
	OP80_DLY_BEF_MEAS : INT;
	OP80_VERT_SERVO_WORK_POS : REAL;
	OP80_VERT_SERVO_SFE_WORK_POS : REAL;	
END_VAR

// ---- POUs/Programs/OP90/OP90_HMI_GVL.TcGVL
//{attribute 'qualified_only'}
VAR_GLOBAL
	
//	SERVO
	OP90_SRV_HORZ_CNTRL						: Servo_Control;
	OP90_SRV_LH_VERT_CNTRL                  : Servo_Control;
	OP90_SRV_RH_VERT_CNTRL                  : Servo_Control;
	OP90_STP_LH_ROTRY_CNTRL					: SERVO_Control;
	OP90_STP_RH_ROTRY_CNTRL					: SERVO_Control;
	OP90_SERVO_GUIDE_CNTRL					: Servo_Control;
	OP90_SRV_LH_CNVY_CNTRL					: Servo_Control;
	OP90_SRV_RH_CNVY_CNTRL                  : Servo_Control;
//LREAL	
	OP90_SERVO_ACTUAL_POS					: LREAL;
//REAL
	OP90_TRGT_POS							: REAL;
	OP90_TRGT_VEL							: REAL;
// INT
	OP90_CYL_NUM							: INT;
	OP90_SERVO_NUM							: INT;
	OP90_AUTO_STATUS_MES					: INT;	
// BOOL
	OP90_JOG_POS							: BOOL;
	OP90_JOG_NEG							: BOOL;	
	OP90_HOME								: BOOL;
	OP90_WORK								: BOOL;
	OP90_SET_HME							: BOOL;
	OP90_MOVE_TARGT							: BOOL;
	OP90_SERVO_FAULT						: BOOL;
	OP90_HOME_REFERENCE						: BOOL;
	OP90_M_SERVO_ENABLE						: BOOL;
	OP90_HOMING_STRT						: BOOL;
END_VAR
VAR_GLOBAL PERSISTENT
// LREAL
	OP90_SRV_HORZ_WRK_MM					: LREAL;
	OP90_SRV_HORZ_HME_MM					: LREAL;
	OP90_SRV_VERT_LH_HME_MM					: LREAL;
	OP90_SRV_VERT_LH_PCKWRK_MM				: LREAL;
    OP90_SRV_VERT_LH_SPLCWRK_MM         	: LREAL;
    OP90_SRV_VERT_LH_PLCWRK_MM          	: LREAL;
	OP90_SRV_VERT_RH_HME_MM					: LREAL;
	OP90_SRV_VERT_RH_PCKWRK_MM		    	: LREAL;
    OP90_SRV_VERT_RH_SPLCWRK_MM         	: LREAL;
    OP90_SRV_VERT_RH_PLCWRK_MM          	: LREAL;
	OP90_STP_ROTRY_LH_HME_MM				: LREAL;
	OP90_STP_ROTRY_RH_HME_MM				: LREAL;
	OP90_STP_ROTRY_LH_WRK_MM				: LREAL;
	OP90_STP_ROTRY_RH_WRK_MM            	: LREAL;
	OP90_SRV_LIMIT							: OP90_SERVO_LIMIT;
END_VAR

// ---- POUs/Programs/OP90/OP90_VARIABLE.TcGVL
VAR_GLOBAL
// MODE_BLOCK
	OP90_MODE_BLOCK							:Mode_Selection_Block1;
	MACHINE_1S 								: BOOL;
	MACHINE_BLINK							: BOOL;
	OP90_MODE_WORD							: INT;
	OP90_STRT_PB							: BOOL;
	OP90_RESET_PB							: BOOL;
	OP90_AUTO_SELECTED						: BOOL;
	OP90_MANUAL_SELECTED					: BOOL;
	OP90_STEP_SELECTED						: BOOL;
	OP90_AUTO_RUNNING						: BOOL;
	OP90_STEP_RUNNING						: BOOL;
	OP90_START_ENABLE						: BOOL;
	OP90_MACHINE_STOP						: BOOL;
	OP90_ERR								: BOOL;	
	OP90_OPERATION_ENABLE					: BOOL;
// FUNTIONAL BLOCK
							(*CYLINDER*)
	OP90_LH_GRIPPER							: Cylinder_Block;
	OP90_RH_GRIPPER							: Cylinder_Block;	
	OP90_POS1_LCK_CYL						: Cylinder_Block;
	OP90_POS2_LCK_CYL						: Cylinder_Block;
	OP90_POS_SLIDE_CYL						: Cylinder_Block;	
	OP90_SUP_HORZP1_CYL						: Cylinder_Block;
	OP90_SUP_VERTP1_CYL                     : Cylinder_Block;
	OP90_SUP_HORZP2_CYL	                    : Cylinder_Block; 
	OP90_SUP_VERTP2_CYL	                    : Cylinder_Block; 
	OP90_LH_REJP1_CYL						: Cylinder_Block;
	OP90_RH_REJP1_CYL                       : Cylinder_Block;
	OP90_LH_REJP2_CYL                       : Cylinder_Block;
	OP90_RH_REJP2_CYL                       : Cylinder_Block;
							(*SERVO*)
	OP90_SRVO_HORZ							: AXIS_REF;						
	OP90_SRVO_LH_VERT						: AXIS_REF;	
	OP90_SRVO_RH_VERT						: AXIS_REF;
	OP90_STP_LH_ROTRY						: AXIS_REF;
	OP90_STP_RH_ROTRY						: AXIS_REF;
	OP90_GUID_SERV							: AXIS_REF;
	OP90_SRV_CNVY_LH						: AXIS_REF;
	OP90_SRV_CNVY_RH						: AXIS_REF;						
	OP90_SRV_HORZ							: FB_Axis_FESTO;
	OP90_SRV_LH_VERT						: FB_Axis_FESTO;
	OP90_SRV_RH_VERT						: FB_Axis_FESTO;
	OP90_GUIDE_SERVO						: FB_Axis_FESTO;
	OP90_LH_SRV_ROTRY						: FB_Axis_FESTO;
	OP90_RH_SRV_ROTRY						: FB_Axis_FESTO;
	OP90_LH_CNVY							: FB_Axis;
	OP90_RH_CNVY							: FB_Axis;
	OP90_SRV_HORZ_STATUS					: stManualModeAxis;
	OP90_SRV_LH_VERT_STATUS                 : stManualModeAxis;
	OP90_SRV_RH_VERT_STATUS                 : stManualModeAxis;
	OP90_STP_LH_ROTRY_STATUS				: stManualModeAxis;
	OP90_STP_RH_ROTRY_STATUS				: stManualModeAxis;
	OP90_GIUDE_SER_STATUS					: stManualModeAxis;
	OP90_SRV_LH_CNVY_STATUS					: stManualModeAxis;
	OP90_SRV_RH_CNVY_STATUS                 : stManualModeAxis;
	
// HOMING 
//BOOL
	OP90_ALL_HOME							: BOOL;
	OP90_START_HOMNG								: BOOL;
	OP90_LH_GRP_HOMING1						: BOOL;
	OP90_RH_GRP_HOMING1						: BOOL;
	OP90_VERT_LHSERV_HOMG1					: BOOL;
	OP90_VERT_RHSERV_HOMG1					: BOOL;
	OP90_LH_GRP_SNR1						: BOOL;
	OP90_HORZ_SERV_HOMING1					: BOOL;
	OP90_VERT_SERVO_HOME					: BOOL;
	OP90_SUP_VERTP1_CYL_HOME1				: BOOL;
	OP90_SUP_HORZP1_CYL_HOME1				: BOOL;
	OP90_SUP_VERTP2_CYL_HOME1				: BOOL;
	OP90_SUP_HORZP2_CYL_HOME1				: BOOL;
	OP90_SUP_VERT_CYL_SNR1					: BOOL;
// INT
	OP90_HME_STP_NO							: INT;
	OP10A_HME_STP_NO						: INT;
	OP10B_HME_STP_NO						: INT;	
//MANUAL
	OP90A_CYLINDER_ERR						: WORD;

								(*SERVO*)

	
	
// AUTO	
	OP90_STN_ENABLE							: BOOL;
	OP90_LH_GRP_BYPASS						: BOOL;
	OP90_RH_GRP_BYPASS						: BOOL;
	OP90_pick_ready							: BOOL;
	OP90_pick_done_7_89						: BOOL;	
	OP90_pick_done_6_38						: BOOL;	
								(*CYLINDER*)

	OP90_A_MVR_SUP_HORZP1_WRK				: BOOL;
	OP90_A_MVR_SUP_HORZP1_HME				: BOOL;
	OP90_A_MVR_SUP_HORZP2_HME				: BOOL;
	OP90_A_MVR_SUP_HORZP2_WRK				: BOOL;
	OP90_A_MVR_SUP_VERTP1_HME				: BOOL;
	OP90_A_MVR_SUP_VERTP1_WRK				: BOOL;
	OP90_A_MVR_SUP_VERTP2_HME				: BOOL;
	OP90_A_MVR_SUP_VERTP2_WRK				: BOOL;
	OP90_POS2_V7_89							: BOOL;				// BASED ON THE MODEL SELECTION OP90_POS1_V6_3 R POS 2 IS CHOOSEN FROM RECEIPE
	OP90_POS1_V6_3							: BOOL;	
	OP90_A_RH_GRP_AUTCMD2					: BOOL;
	OP90_A_RH_GRP_AUTCMD1					: BOOL;
	OP90_A_LH_GRP_AUTCMD2					: BOOL;
	OP90_A_LH_GRP_AUTCMD1					: BOOL;
	OP90_A_LH_REJP1_HOME					: BOOL;
	OP90_A_RH_REJP1_HOME					: BOOL;
	OP90_A_LH_REJP1_WORK					: BOOL;
	OP90_A_RH_REJP1_WORK					: BOOL;
	OP90_A_LH_REJP2_HOME					: BOOL;
	OP90_A_RH_REJP2_HOME					: BOOL;
	OP90_A_LH_REJP2_WORK					: BOOL;
	OP90_A_RH_REJP2_WORK					: BOOL;	
	
	
	
	
	
								(*SERVO*)
// BOOL
	OP90_A_SRV_HORZ_WRK						: BOOL;
	OP90_A_SRV_HORZ_HME						: BOOL;	
	OP90_A_SRV_LHVERT_HME					: BOOL;	
	OP90_A_SRV_LHVERT_PCKWRK				: BOOL;
	OP90_A_SRV_LHVERT_SPLCWRK				: BOOL;
	OP90_A_SRV_LHVERT_PLCWRK				: BOOL;
	OP90_A_SRV_RHVERT_HME					: BOOL;	
	OP90_A_SRV_RHVERT_PCKWRK				: BOOL;
	OP90_A_SRV_RHVERT_SPLCWRK				: BOOL;
	OP90_A_SRV_RHVERT_PLCWRK				: BOOL;
	OP90_A_SRV_LH_ROTRY_WRK					: BOOL;
	OP90_A_SRV_LH_ROTRY_HME					: BOOL;	
	OP90_A_SRV_RH_ROTRY_WRK					: BOOL;	
	OP90_A_SRV_RH_ROTRY_HME					: BOOL;	
	
	OP90_SRV_LH_VRT_HME_FB					: BOOL;
	OP90_SRV_RH_VRT_HME_FB					: BOOL;
	OP90_SRV_HORZ_HME_FB					: BOOL;
	OP90_SRV_HORZ_WRK_FB					: BOOL;
	OP90_SRV_LH_VRT_PCKWRK_FB				: BOOL;
	OP90_SRV_RH_VRT_PCKWRK_FB				: BOOL;
	OP90_SRV_LH_VRT_SPLCWRK_FB				: BOOL;
	OP90_SRV_RH_VRT_SPLCWRK_FB				: BOOL;
	OP90_SRV_LH_VRT_PLCWRK_FB				: BOOL;	
	OP90_SRV_RH_VRT_PLCWRK_FB				: BOOL;
	OP90_STP_LH_ROTY_HME_FB					: BOOL;
	OP90_STP_LH_ROTY_WRK_FB					: BOOL;
	OP90_STP_RH_ROTY_HME_FB					: BOOL;
	OP90_STP_RH_ROTY_WRK_FB					: BOOL;
	OP90_SRV_HORZ_ZERO_FB					: BOOL;
	OP90_SRV_LH_VRT_ZERO_FB					: BOOL;
	OP90_SRV_RH_VRT_ZERO_FB					: BOOL;
	OP90_VERT_SRV_SAFE_ZONE					: BOOL;
	
								(*CAMERA*)
	OP90_CAMERA_TRIGGER						: BOOL;								
	OP90_LH_CMR_OK							: BOOL;
	OP90_LH_CMR_NOK							: BOOL;	
	OP90_RH_CMR_OK							: BOOL;
	OP90_RH_CMR_NOK							: BOOL;	
	//OP90_Camera_Done						: BOOL;

	
	
//XTS
	OP90_MVR_LH_CMPNOK						: BOOL;
	OP90_MVR_RH_CMPNOK						: BOOL;	

// WILL BE DELETED 
MACHINE_ERR		: BOOL;
MACHINE_AUTO    : BOOL;
MACHINE_MANUAL	: BOOL;

//Camera GVLs
	OP90_LH_Camera_Trigger		      : BOOL;
	OP90_LH_Camera_Job_Change_start   : BOOL;
	OP90_LH_Camera_Error			  : BOOL;
	OP90_LH_Camera_Ready			  : BOOL;
	OP90_LH_Camera_Online			  : BOOL;	
	OP90_LH_Job_Change_Complete		    : BOOL;
	OP90_LH_Job_Change_Error   		    : BOOL;
	OP90_LH_Picture_Taken      		    : BOOL;
	OP90_LH_Error_status				: STRING;
	OP90_LH_Target_Job_ID				: UINT;
	OP90_LH_Loaded_Job_ID		    	: UINT;

	OP90_RH_Camera_Trigger		      : BOOL;
	OP90_RH_Camera_Job_Change_start   : BOOL;
	OP90_RH_Camera_Error			  : BOOL;
	OP90_RH_Camera_Ready			  : BOOL;
	OP90_RH_Camera_Online			  : BOOL;	
	OP90_RH_Job_Change_Complete		    : BOOL;
	OP90_RH_Job_Change_Error   		    : BOOL;
	OP90_RH_Picture_Taken      		    : BOOL;
	OP90_RH_Error_status				: STRING;
	OP90_RH_Target_Job_ID				: UINT;
	OP90_RH_Loaded_Job_ID		    	: UINT;

	OP90_Camera_Trigger_Ack: BOOL;
	OP90_Miss_Trigger: BOOL;
	OP90_LH_Camera_OK  : BOOL;
	OP90_LH_Camera_NOK : BOOL;
	OP90_RH_Camera_OK  : BOOL;
	OP90_RH_Camera_NOK : BOOL;
	OP90_Camera_Done	: BOOL;	
	
END_VAR

VAR_GLOBAL PERSISTENT
// AUTO
							(*CYLINDER*)
	OP90_LH_CMP_PICKED						: BOOL;
	OP90_RH_CMP_PICKED						: BOOL;
END_VAR

// ---- POUs/GENERAL/Robot_232_Comm_Prgrm.TcPOU
PROGRAM Robot_232_Comm_Prgrm
VAR
	BioMetric_In_All AT %I*: EL6inData22B;
	BioMetric_Out_All AT %Q*: EL6outData22B;	
	Bio_Metric		:SerialLineControl;
	Error			: BOOL;
	Error_ID		: ComError_t;
	
	Comm_Delay   : TON;
	Initial		 : BOOL;
	bSendDataRisingEdge: R_TRIG;
	bSendData: BOOL;
	fbSendString : SendString;
	sSendStringData : STRING;
	bSendBusy  : BOOL;
	sSendError : ComError_t;
END_VAR

Comm_Delay(IN:= NOT Initial,PT:=T#15S);

OP10_ROBO();
OP160_Robo_Byte_Mapping();
OP160_Robo_Inputs();
OP120_Robo_Byte_Mapping();
OP120_Robo_Inputs();

IF Comm_Delay.Q THEN
	Initial:=1;
END_IF

IF Initial THEN
	Bio_Metric(Mode:= , 
	pComIn:=(ADR(BioMetric_In_All)) , 
	pComOut:=(ADR(BioMetric_Out_All)) , 
	SizeComIn:=SIZEOF(BioMetric_In_All), 
	Error=> Error, 
	ErrorID=>Error_ID , 
	TxBuffer:= SerialComm.TxBuffer_1, 
	RxBuffer:=SerialComm.RxBuffer_1 );
END_IF

bSendDataRisingEdge(CLK:=bSendData);

IF bSendDataRisingEdge.Q THEN

	fbSendString(SendString:= sSendStringData,
				TXBuffer:=SerialComm.TxBuffer_1,
				Busy=>bSendBusy,
				Error=>sSendError
				);

END_IF

END_PROGRAM

// ---- POUs/Error.TcPOU
PROGRAM Error
VAR
	
Alarm: FB_TcEventLogger;
	bint:BOOL;
	Error:  ARRAY [0..2001] OF FB_TcAlarm;
	
	i:INT;
	j:int;
	
	bdone: BOOL;
	
	Bin1:BOOL;
	Bin2:BOOL;
	Bin3:BOOL;
	Bin4:BOOL;
	Bin5:BOOL;
	Bin6:BOOL;
	Bin7:BOOL;
	temp: BOOL;
	
	bInit: BOOL;
	bRaise: BOOL;
	bclearA: BOOL;
END_VAR


IF NOT bint THEN
	bint:=TRUE;
Error[1].CreateEx(TC_Events.Error.Error1,FALSE,0);
Error[2].CreateEx(TC_Events.Error.Error2,FALSE,0);
Error[3].CreateEx(TC_Events.Error.Error3,FALSE,0);
Error[4].CreateEx(TC_Events.Error.Error4,FALSE,0);
Error[5].CreateEx(TC_Events.Error.Error5,FALSE,0);
Error[6].CreateEx(TC_Events.Error.Error6,FALSE,0);
Error[7].CreateEx(TC_Events.Error.Error7,FALSE,0);
Error[8].CreateEx(TC_Events.Error.Error8,FALSE,0);
Error[9].CreateEx(TC_Events.Error.Error9,FALSE,0);
Error[10].CreateEx(TC_Events.Error.Error10,FALSE,0);
Error[11].CreateEx(TC_Events.Error.Error11,FALSE,0);
Error[12].CreateEx(TC_Events.Error.Error12,FALSE,0);
Error[13].CreateEx(TC_Events.Error.Error13,FALSE,0);
Error[14].CreateEx(TC_Events.Error.Error14,FALSE,0);
Error[15].CreateEx(TC_Events.Error.Error15,FALSE,0);
Error[16].CreateEx(TC_Events.Error.Error16,FALSE,0);
Error[17].CreateEx(TC_Events.Error.Error17,FALSE,0);
Error[18].CreateEx(TC_Events.Error.Error18,FALSE,0);
Error[19].CreateEx(TC_Events.Error.Error19,FALSE,0);
Error[20].CreateEx(TC_Events.Error.Error20,FALSE,0);
Error[21].CreateEx(TC_Events.Error.Error21,FALSE,0);
Error[22].CreateEx(TC_Events.Error.Error22,FALSE,0);
Error[23].CreateEx(TC_Events.Error.Error23,FALSE,0);
Error[24].CreateEx(TC_Events.Error.Error24,FALSE,0);
Error[25].CreateEx(TC_Events.Error.Error25,FALSE,0);
Error[26].CreateEx(TC_Events.Error.Error26,FALSE,0);
Error[27].CreateEx(TC_Events.Error.Error27,FALSE,0);
Error[28].CreateEx(TC_Events.Error.Error28,FALSE,0);
Error[29].CreateEx(TC_Events.Error.Error29,FALSE,0);
Error[30].CreateEx(TC_Events.Error.Error30,FALSE,0);
Error[31].CreateEx(TC_Events.Error.Error31,FALSE,0);
Error[32].CreateEx(TC_Events.Error.Error32,FALSE,0);
Error[33].CreateEx(TC_Events.Error.Error33,FALSE,0);
Error[34].CreateEx(TC_Events.Error.Error34,FALSE,0);
Error[35].CreateEx(TC_Events.Error.Error35,FALSE,0);
Error[36].CreateEx(TC_Events.Error.Error36,FALSE,0);
Error[37].CreateEx(TC_Events.Error.Error37,FALSE,0);
Error[38].CreateEx(TC_Events.Error.Error38,FALSE,0);
Error[39].CreateEx(TC_Events.Error.Error39,FALSE,0);
Error[40].CreateEx(TC_Events.Error.Error40,FALSE,0);
Error[41].CreateEx(TC_Events.Error.Error41,FALSE,0);
Error[42].CreateEx(TC_Events.Error.Error42,FALSE,0);
Error[43].CreateEx(TC_Events.Error.Error43,FALSE,0);
Error[44].CreateEx(TC_Events.Error.Error44,FALSE,0);
Error[45].CreateEx(TC_Events.Error.Error45,FALSE,0);
Error[46].CreateEx(TC_Events.Error.Error46,FALSE,0);
Error[47].CreateEx(TC_Events.Error.Error47,FALSE,0);
Error[48].CreateEx(TC_Events.Error.Error48,FALSE,0);
Error[49].CreateEx(TC_Events.Error.Error49,FALSE,0);
Error[50].CreateEx(TC_Events.Error.Error50,FALSE,0);
Error[51].CreateEx(TC_Events.Error.Error51,FALSE,0);
Error[52].CreateEx(TC_Events.Error.Error52,FALSE,0);
Error[53].CreateEx(TC_Events.Error.Error53,FALSE,0);
Error[54].CreateEx(TC_Events.Error.Error54,FALSE,0);
Error[55].CreateEx(TC_Events.Error.Error55,FALSE,0);
Error[56].CreateEx(TC_Events.Error.Error56,FALSE,0);
Error[57].CreateEx(TC_Events.Error.Error57,FALSE,0);
Error[58].CreateEx(TC_Events.Error.Error58,FALSE,0);
Error[59].CreateEx(TC_Events.Error.Error59,FALSE,0);
Error[60].CreateEx(TC_Events.Error.Error60,FALSE,0);
Error[61].CreateEx(TC_Events.Error.Error61,FALSE,0);
Error[62].CreateEx(TC_Events.Error.Error62,FALSE,0);
Error[63].CreateEx(TC_Events.Error.Error63,FALSE,0);
Error[64].CreateEx(TC_Events.Error.Error64,FALSE,0);
Error[65].CreateEx(TC_Events.Error.Error65,FALSE,0);
Error[66].CreateEx(TC_Events.Error.Error66,FALSE,0);
Error[67].CreateEx(TC_Events.Error.Error67,FALSE,0);
Error[68].CreateEx(TC_Events.Error.Error68,FALSE,0);
Error[69].CreateEx(TC_Events.Error.Error69,FALSE,0);
Error[70].CreateEx(TC_Events.Error.Error70,FALSE,0);
Error[71].CreateEx(TC_Events.Error.Error71,FALSE,0);
Error[72].CreateEx(TC_Events.Error.Error72,FALSE,0);
Error[73].CreateEx(TC_Events.Error.Error73,FALSE,0);
Error[74].CreateEx(TC_Events.Error.Error74,FALSE,0);
Error[75].CreateEx(TC_Events.Error.Error75,FALSE,0);
Error[76].CreateEx(TC_Events.Error.Error76,FALSE,0);
Error[77].CreateEx(TC_Events.Error.Error77,FALSE,0);
Error[78].CreateEx(TC_Events.Error.Error78,FALSE,0);
Error[79].CreateEx(TC_Events.Error.Error79,FALSE,0);
Error[80].CreateEx(TC_Events.Error.Error80,FALSE,0);
Error[81].CreateEx(TC_Events.Error.Error81,FALSE,0);
Error[82].CreateEx(TC_Events.Error.Error82,FALSE,0);
Error[83].CreateEx(TC_Events.Error.Error83,FALSE,0);
Error[84].CreateEx(TC_Events.Error.Error84,FALSE,0);
Error[85].CreateEx(TC_Events.Error.Error85,FALSE,0);
Error[86].CreateEx(TC_Events.Error.Error86,FALSE,0);
Error[87].CreateEx(TC_Events.Error.Error87,FALSE,0);
Error[88].CreateEx(TC_Events.Error.Error88,FALSE,0);
Error[89].CreateEx(TC_Events.Error.Error89,FALSE,0);
Error[90].CreateEx(TC_Events.Error.Error90,FALSE,0);
Error[91].CreateEx(TC_Events.Error.Error91,FALSE,0);
Error[92].CreateEx(TC_Events.Error.Error92,FALSE,0);
Error[93].CreateEx(TC_Events.Error.Error93,FALSE,0);
Error[94].CreateEx(TC_Events.Error.Error94,FALSE,0);
Error[95].CreateEx(TC_Events.Error.Error95,FALSE,0);
Error[96].CreateEx(TC_Events.Error.Error96,FALSE,0);
Error[97].CreateEx(TC_Events.Error.Error97,FALSE,0);
Error[98].CreateEx(TC_Events.Error.Error98,FALSE,0);
Error[99].CreateEx(TC_Events.Error.Error99,FALSE,0);
Error[100].CreateEx(TC_Events.Error.Error100,FALSE,0);
Error[101].CreateEx(TC_Events.Error.Error101,FALSE,0);
Error[102].CreateEx(TC_Events.Error.Error102,FALSE,0);
Error[103].CreateEx(TC_Events.Error.Error103,FALSE,0);
Error[104].CreateEx(TC_Events.Error.Error104,FALSE,0);
Error[105].CreateEx(TC_Events.Error.Error105,FALSE,0);
Error[106].CreateEx(TC_Events.Error.Error106,FALSE,0);
Error[107].CreateEx(TC_Events.Error.Error107,FALSE,0);
Error[108].CreateEx(TC_Events.Error.Error108,FALSE,0);
Error[109].CreateEx(TC_Events.Error.Error109,FALSE,0);
Error[110].CreateEx(TC_Events.Error.Error110,FALSE,0);
Error[111].CreateEx(TC_Events.Error.Error111,FALSE,0);
Error[112].CreateEx(TC_Events.Error.Error112,FALSE,0);
Error[113].CreateEx(TC_Events.Error.Error113,FALSE,0);
Error[114].CreateEx(TC_Events.Error.Error114,FALSE,0);
Error[115].CreateEx(TC_Events.Error.Error115,FALSE,0);
Error[116].CreateEx(TC_Events.Error.Error116,FALSE,0);
Error[117].CreateEx(TC_Events.Error.Error117,FALSE,0);
Error[118].CreateEx(TC_Events.Error.Error118,FALSE,0);
Error[119].CreateEx(TC_Events.Error.Error119,FALSE,0);
Error[120].CreateEx(TC_Events.Error.Error120,FALSE,0);
Error[121].CreateEx(TC_Events.Error.Error121,FALSE,0);
Error[122].CreateEx(TC_Events.Error.Error122,FALSE,0);
Error[123].CreateEx(TC_Events.Error.Error123,FALSE,0);
Error[124].CreateEx(TC_Events.Error.Error124,FALSE,0);
Error[125].CreateEx(TC_Events.Error.Error125,FALSE,0);
Error[126].CreateEx(TC_Events.Error.Error126,FALSE,0);
Error[127].CreateEx(TC_Events.Error.Error127,FALSE,0);
Error[128].CreateEx(TC_Events.Error.Error128,FALSE,0);
Error[129].CreateEx(TC_Events.Error.Error129,FALSE,0);
Error[130].CreateEx(TC_Events.Error.Error130,FALSE,0);
Error[131].CreateEx(TC_Events.Error.Error131,FALSE,0);
Error[132].CreateEx(TC_Events.Error.Error132,FALSE,0);
Error[133].CreateEx(TC_Events.Error.Error133,FALSE,0);
Error[134].CreateEx(TC_Events.Error.Error134,FALSE,0);
Error[135].CreateEx(TC_Events.Error.Error135,FALSE,0);
Error[136].CreateEx(TC_Events.Error.Error136,FALSE,0);
Error[137].CreateEx(TC_Events.Error.Error137,FALSE,0);
Error[138].CreateEx(TC_Events.Error.Error138,FALSE,0);
Error[139].CreateEx(TC_Events.Error.Error139,FALSE,0);
Error[140].CreateEx(TC_Events.Error.Error140,FALSE,0);
Error[141].CreateEx(TC_Events.Error.Error141,FALSE,0);
Error[142].CreateEx(TC_Events.Error.Error142,FALSE,0);
Error[143].CreateEx(TC_Events.Error.Error143,FALSE,0);
Error[144].CreateEx(TC_Events.Error.Error144,FALSE,0);
Error[145].CreateEx(TC_Events.Error.Error145,FALSE,0);
Error[146].CreateEx(TC_Events.Error.Error146,FALSE,0);
Error[147].CreateEx(TC_Events.Error.Error147,FALSE,0);
Error[148].CreateEx(TC_Events.Error.Error148,FALSE,0);
Error[149].CreateEx(TC_Events.Error.Error149,FALSE,0);
Error[150].CreateEx(TC_Events.Error.Error150,FALSE,0);
Error[151].CreateEx(TC_Events.Error.Error151,FALSE,0);
Error[152].CreateEx(TC_Events.Error.Error152,FALSE,0);
Error[153].CreateEx(TC_Events.Error.Error153,FALSE,0);
Error[154].CreateEx(TC_Events.Error.Error154,FALSE,0);
Error[155].CreateEx(TC_Events.Error.Error155,FALSE,0);
Error[156].CreateEx(TC_Events.Error.Error156,FALSE,0);
Error[157].CreateEx(TC_Events.Error.Error157,FALSE,0);
Error[158].CreateEx(TC_Events.Error.Error158,FALSE,0);
Error[159].CreateEx(TC_Events.Error.Error159,FALSE,0);
Error[160].CreateEx(TC_Events.Error.Error160,FALSE,0);
Error[161].CreateEx(TC_Events.Error.Error161,FALSE,0);
Error[162].CreateEx(TC_Events.Error.Error162,FALSE,0);
Error[163].CreateEx(TC_Events.Error.Error163,FALSE,0);
Error[164].CreateEx(TC_Events.Error.Error164,FALSE,0);
Error[165].CreateEx(TC_Events.Error.Error165,FALSE,0);
Error[166].CreateEx(TC_Events.Error.Error166,FALSE,0);
Error[167].CreateEx(TC_Events.Error.Error167,FALSE,0);
Error[168].CreateEx(TC_Events.Error.Error168,FALSE,0);
Error[169].CreateEx(TC_Events.Error.Error169,FALSE,0);
Error[170].CreateEx(TC_Events.Error.Error170,FALSE,0);
Error[171].CreateEx(TC_Events.Error.Error171,FALSE,0);
Error[172].CreateEx(TC_Events.Error.Error172,FALSE,0);
Error[173].CreateEx(TC_Events.Error.Error173,FALSE,0);
Error[174].CreateEx(TC_Events.Error.Error174,FALSE,0);
Error[175].CreateEx(TC_Events.Error.Error175,FALSE,0);
Error[176].CreateEx(TC_Events.Error.Error176,FALSE,0);
Error[177].CreateEx(TC_Events.Error.Error177,FALSE,0);
Error[178].CreateEx(TC_Events.Error.Error178,FALSE,0);
Error[179].CreateEx(TC_Events.Error.Error179,FALSE,0);
Error[180].CreateEx(TC_Events.Error.Error180,FALSE,0);
Error[181].CreateEx(TC_Events.Error.Error181,FALSE,0);
Error[182].CreateEx(TC_Events.Error.Error182,FALSE,0);
Error[183].CreateEx(TC_Events.Error.Error183,FALSE,0);
Error[184].CreateEx(TC_Events.Error.Error184,FALSE,0);
Error[185].CreateEx(TC_Events.Error.Error185,FALSE,0);
Error[186].CreateEx(TC_Events.Error.Error186,FALSE,0);
Error[187].CreateEx(TC_Events.Error.Error187,FALSE,0);
Error[188].CreateEx(TC_Events.Error.Error188,FALSE,0);
Error[189].CreateEx(TC_Events.Error.Error189,FALSE,0);
Error[190].CreateEx(TC_Events.Error.Error190,FALSE,0);
Error[191].CreateEx(TC_Events.Error.Error191,FALSE,0);
Error[192].CreateEx(TC_Events.Error.Error192,FALSE,0);
Error[193].CreateEx(TC_Events.Error.Error193,FALSE,0);
Error[194].CreateEx(TC_Events.Error.Error194,FALSE,0);
Error[195].CreateEx(TC_Events.Error.Error195,FALSE,0);
Error[196].CreateEx(TC_Events.Error.Error196,FALSE,0);
Error[197].CreateEx(TC_Events.Error.Error197,FALSE,0);
Error[198].CreateEx(TC_Events.Error.Error198,FALSE,0);
Error[199].CreateEx(TC_Events.Error.Error199,FALSE,0);
Error[200].CreateEx(TC_Events.Error.Error200,FALSE,0);
Error[201].CreateEx(TC_Events.Error.Error201,FALSE,0);
Error[202].CreateEx(TC_Events.Error.Error202,FALSE,0);
Error[203].CreateEx(TC_Events.Error.Error203,FALSE,0);
Error[204].CreateEx(TC_Events.Error.Error204,FALSE,0);
Error[205].CreateEx(TC_Events.Error.Error205,FALSE,0);
Error[206].CreateEx(TC_Events.Error.Error206,FALSE,0);
Error[207].CreateEx(TC_Events.Error.Error207,FALSE,0);
Error[208].CreateEx(TC_Events.Error.Error208,FALSE,0);
Error[209].CreateEx(TC_Events.Error.Error209,FALSE,0);
Error[210].CreateEx(TC_Events.Error.Error210,FALSE,0);
Error[211].CreateEx(TC_Events.Error.Error211,FALSE,0);
Error[212].CreateEx(TC_Events.Error.Error212,FALSE,0);
Error[213].CreateEx(TC_Events.Error.Error213,FALSE,0);
Error[214].CreateEx(TC_Events.Error.Error214,FALSE,0);
Error[215].CreateEx(TC_Events.Error.Error215,FALSE,0);
Error[216].CreateEx(TC_Events.Error.Error216,FALSE,0);
Error[217].CreateEx(TC_Events.Error.Error217,FALSE,0);
Error[218].CreateEx(TC_Events.Error.Error218,FALSE,0);
Error[219].CreateEx(TC_Events.Error.Error219,FALSE,0);
Error[220].CreateEx(TC_Events.Error.Error220,FALSE,0);
Error[221].CreateEx(TC_Events.Error.Error221,FALSE,0);
Error[222].CreateEx(TC_Events.Error.Error222,FALSE,0);
Error[223].CreateEx(TC_Events.Error.Error223,FALSE,0);
Error[224].CreateEx(TC_Events.Error.Error224,FALSE,0);
Error[225].CreateEx(TC_Events.Error.Error225,FALSE,0);
Error[226].CreateEx(TC_Events.Error.Error226,FALSE,0);
Error[227].CreateEx(TC_Events.Error.Error227,FALSE,0);
Error[228].CreateEx(TC_Events.Error.Error228,FALSE,0);
Error[229].CreateEx(TC_Events.Error.Error229,FALSE,0);
Error[230].CreateEx(TC_Events.Error.Error230,FALSE,0);
Error[231].CreateEx(TC_Events.Error.Error231,FALSE,0);
Error[232].CreateEx(TC_Events.Error.Error232,FALSE,0);
Error[233].CreateEx(TC_Events.Error.Error233,FALSE,0);
Error[234].CreateEx(TC_Events.Error.Error234,FALSE,0);
Error[235].CreateEx(TC_Events.Error.Error235,FALSE,0);
Error[236].CreateEx(TC_Events.Error.Error236,FALSE,0);
Error[237].CreateEx(TC_Events.Error.Error237,FALSE,0);
Error[238].CreateEx(TC_Events.Error.Error238,FALSE,0);
Error[239].CreateEx(TC_Events.Error.Error239,FALSE,0);
Error[240].CreateEx(TC_Events.Error.Error240,FALSE,0);
Error[241].CreateEx(TC_Events.Error.Error241,FALSE,0);
Error[242].CreateEx(TC_Events.Error.Error242,FALSE,0);
Error[243].CreateEx(TC_Events.Error.Error243,FALSE,0);
Error[244].CreateEx(TC_Events.Error.Error244,FALSE,0);
Error[245].CreateEx(TC_Events.Error.Error245,FALSE,0);
Error[246].CreateEx(TC_Events.Error.Error246,FALSE,0);
Error[247].CreateEx(TC_Events.Error.Error247,FALSE,0);
Error[248].CreateEx(TC_Events.Error.Error248,FALSE,0);
Error[249].CreateEx(TC_Events.Error.Error249,FALSE,0);
Error[250].CreateEx(TC_Events.Error.Error250,FALSE,0);
Error[251].CreateEx(TC_Events.Error.Error251,FALSE,0);
Error[252].CreateEx(TC_Events.Error.Error252,FALSE,0);
Error[253].CreateEx(TC_Events.Error.Error253,FALSE,0);
Error[254].CreateEx(TC_Events.Error.Error254,FALSE,0);
Error[255].CreateEx(TC_Events.Error.Error255,FALSE,0);
Error[256].CreateEx(TC_Events.Error.Error256,FALSE,0);
Error[257].CreateEx(TC_Events.Error.Error257,FALSE,0);
Error[258].CreateEx(TC_Events.Error.Error258,FALSE,0);
Error[259].CreateEx(TC_Events.Error.Error259,FALSE,0);
Error[260].CreateEx(TC_Events.Error.Error260,FALSE,0);
Error[261].CreateEx(TC_Events.Error.Error261,FALSE,0);
Error[262].CreateEx(TC_Events.Error.Error262,FALSE,0);
Error[263].CreateEx(TC_Events.Error.Error263,FALSE,0);
Error[264].CreateEx(TC_Events.Error.Error264,FALSE,0);
Error[265].CreateEx(TC_Events.Error.Error265,FALSE,0);
Error[266].CreateEx(TC_Events.Error.Error266,FALSE,0);
Error[267].CreateEx(TC_Events.Error.Error267,FALSE,0);
Error[268].CreateEx(TC_Events.Error.Error268,FALSE,0);
Error[269].CreateEx(TC_Events.Error.Error269,FALSE,0);
Error[270].CreateEx(TC_Events.Error.Error270,FALSE,0);
Error[271].CreateEx(TC_Events.Error.Error271,FALSE,0);
Error[272].CreateEx(TC_Events.Error.Error272,FALSE,0);
Error[273].CreateEx(TC_Events.Error.Error273,FALSE,0);
Error[274].CreateEx(TC_Events.Error.Error274,FALSE,0);
Error[275].CreateEx(TC_Events.Error.Error275,FALSE,0);
Error[276].CreateEx(TC_Events.Error.Error276,FALSE,0);
Error[277].CreateEx(TC_Events.Error.Error277,FALSE,0);
Error[278].CreateEx(TC_Events.Error.Error278,FALSE,0);
Error[279].CreateEx(TC_Events.Error.Error279,FALSE,0);
Error[280].CreateEx(TC_Events.Error.Error280,FALSE,0);
Error[281].CreateEx(TC_Events.Error.Error281,FALSE,0);
Error[282].CreateEx(TC_Events.Error.Error282,FALSE,0);
Error[283].CreateEx(TC_Events.Error.Error283,FALSE,0);
Error[284].CreateEx(TC_Events.Error.Error284,FALSE,0);
Error[285].CreateEx(TC_Events.Error.Error285,FALSE,0);
Error[286].CreateEx(TC_Events.Error.Error286,FALSE,0);
Error[287].CreateEx(TC_Events.Error.Error287,FALSE,0);
Error[288].CreateEx(TC_Events.Error.Error288,FALSE,0);
Error[289].CreateEx(TC_Events.Error.Error289,FALSE,0);
Error[290].CreateEx(TC_Events.Error.Error290,FALSE,0);
Error[291].CreateEx(TC_Events.Error.Error291,FALSE,0);
Error[292].CreateEx(TC_Events.Error.Error292,FALSE,0);
Error[293].CreateEx(TC_Events.Error.Error293,FALSE,0);
Error[294].CreateEx(TC_Events.Error.Error294,FALSE,0);
Error[295].CreateEx(TC_Events.Error.Error295,FALSE,0);
Error[296].CreateEx(TC_Events.Error.Error296,FALSE,0);
Error[297].CreateEx(TC_Events.Error.Error297,FALSE,0);
Error[298].CreateEx(TC_Events.Error.Error298,FALSE,0);
Error[299].CreateEx(TC_Events.Error.Error299,FALSE,0);
Error[300].CreateEx(TC_Events.Error.Error300,FALSE,0);
Error[301].CreateEx(TC_Events.Error.Error301,FALSE,0);
Error[302].CreateEx(TC_Events.Error.Error302,FALSE,0);
Error[303].CreateEx(TC_Events.Error.Error303,FALSE,0);
Error[304].CreateEx(TC_Events.Error.Error304,FALSE,0);
Error[305].CreateEx(TC_Events.Error.Error305,FALSE,0);
Error[306].CreateEx(TC_Events.Error.Error306,FALSE,0);
Error[307].CreateEx(TC_Events.Error.Error307,FALSE,0);
Error[308].CreateEx(TC_Events.Error.Error308,FALSE,0);
Error[309].CreateEx(TC_Events.Error.Error309,FALSE,0);
Error[310].CreateEx(TC_Events.Error.Error310,FALSE,0);
Error[311].CreateEx(TC_Events.Error.Error311,FALSE,0);
Error[312].CreateEx(TC_Events.Error.Error312,FALSE,0);
Error[313].CreateEx(TC_Events.Error.Error313,FALSE,0);
Error[314].CreateEx(TC_Events.Error.Error314,FALSE,0);
Error[315].CreateEx(TC_Events.Error.Error315,FALSE,0);
Error[316].CreateEx(TC_Events.Error.Error316,FALSE,0);
Error[317].CreateEx(TC_Events.Error.Error317,FALSE,0);
Error[318].CreateEx(TC_Events.Error.Error318,FALSE,0);
Error[319].CreateEx(TC_Events.Error.Error319,FALSE,0);
Error[320].CreateEx(TC_Events.Error.Error320,FALSE,0);
Error[321].CreateEx(TC_Events.Error.Error321,FALSE,0);
Error[322].CreateEx(TC_Events.Error.Error322,FALSE,0);
Error[323].CreateEx(TC_Events.Error.Error323,FALSE,0);
Error[324].CreateEx(TC_Events.Error.Error324,FALSE,0);
Error[325].CreateEx(TC_Events.Error.Error325,FALSE,0);
Error[326].CreateEx(TC_Events.Error.Error326,FALSE,0);
Error[327].CreateEx(TC_Events.Error.Error327,FALSE,0);
Error[328].CreateEx(TC_Events.Error.Error328,FALSE,0);
Error[329].CreateEx(TC_Events.Error.Error329,FALSE,0);
Error[330].CreateEx(TC_Events.Error.Error330,FALSE,0);
Error[331].CreateEx(TC_Events.Error.Error331,FALSE,0);
Error[332].CreateEx(TC_Events.Error.Error332,FALSE,0);
Error[333].CreateEx(TC_Events.Error.Error333,FALSE,0);
Error[334].CreateEx(TC_Events.Error.Error334,FALSE,0);
Error[335].CreateEx(TC_Events.Error.Error335,FALSE,0);
Error[336].CreateEx(TC_Events.Error.Error336,FALSE,0);
Error[337].CreateEx(TC_Events.Error.Error337,FALSE,0);
Error[338].CreateEx(TC_Events.Error.Error338,FALSE,0);
Error[339].CreateEx(TC_Events.Error.Error339,FALSE,0);
Error[340].CreateEx(TC_Events.Error.Error340,FALSE,0);
Error[341].CreateEx(TC_Events.Error.Error341,FALSE,0);
Error[342].CreateEx(TC_Events.Error.Error342,FALSE,0);
Error[343].CreateEx(TC_Events.Error.Error343,FALSE,0);
Error[344].CreateEx(TC_Events.Error.Error344,FALSE,0);
Error[345].CreateEx(TC_Events.Error.Error345,FALSE,0);
Error[346].CreateEx(TC_Events.Error.Error346,FALSE,0);
Error[347].CreateEx(TC_Events.Error.Error347,FALSE,0);
Error[348].CreateEx(TC_Events.Error.Error348,FALSE,0);
Error[349].CreateEx(TC_Events.Error.Error349,FALSE,0);
Error[350].CreateEx(TC_Events.Error.Error350,FALSE,0);
Error[351].CreateEx(TC_Events.Error.Error351,FALSE,0);
Error[352].CreateEx(TC_Events.Error.Error352,FALSE,0);
Error[353].CreateEx(TC_Events.Error.Error353,FALSE,0);
Error[354].CreateEx(TC_Events.Error.Error354,FALSE,0);
Error[355].CreateEx(TC_Events.Error.Error355,FALSE,0);
Error[356].CreateEx(TC_Events.Error.Error356,FALSE,0);
Error[357].CreateEx(TC_Events.Error.Error357,FALSE,0);
Error[358].CreateEx(TC_Events.Error.Error358,FALSE,0);
Error[359].CreateEx(TC_Events.Error.Error359,FALSE,0);
Error[360].CreateEx(TC_Events.Error.Error360,FALSE,0);
Error[361].CreateEx(TC_Events.Error.Error361,FALSE,0);
Error[362].CreateEx(TC_Events.Error.Error362,FALSE,0);
Error[363].CreateEx(TC_Events.Error.Error363,FALSE,0);
Error[364].CreateEx(TC_Events.Error.Error364,FALSE,0);
Error[365].CreateEx(TC_Events.Error.Error365,FALSE,0);
Error[366].CreateEx(TC_Events.Error.Error366,FALSE,0);
Error[367].CreateEx(TC_Events.Error.Error367,FALSE,0);
Error[368].CreateEx(TC_Events.Error.Error368,FALSE,0);
Error[369].CreateEx(TC_Events.Error.Error369,FALSE,0);
Error[370].CreateEx(TC_Events.Error.Error370,FALSE,0);
Error[371].CreateEx(TC_Events.Error.Error371,FALSE,0);
Error[372].CreateEx(TC_Events.Error.Error372,FALSE,0);
Error[373].CreateEx(TC_Events.Error.Error373,FALSE,0);
Error[374].CreateEx(TC_Events.Error.Error374,FALSE,0);
Error[375].CreateEx(TC_Events.Error.Error375,FALSE,0);
Error[376].CreateEx(TC_Events.Error.Error376,FALSE,0);
Error[377].CreateEx(TC_Events.Error.Error377,FALSE,0);
Error[378].CreateEx(TC_Events.Error.Error378,FALSE,0);
Error[379].CreateEx(TC_Events.Error.Error379,FALSE,0);
Error[380].CreateEx(TC_Events.Error.Error380,FALSE,0);
Error[381].CreateEx(TC_Events.Error.Error381,FALSE,0);
Error[382].CreateEx(TC_Events.Error.Error382,FALSE,0);
Error[383].CreateEx(TC_Events.Error.Error383,FALSE,0);
Error[384].CreateEx(TC_Events.Error.Error384,FALSE,0);
Error[385].CreateEx(TC_Events.Error.Error385,FALSE,0);
Error[386].CreateEx(TC_Events.Error.Error386,FALSE,0);
Error[387].CreateEx(TC_Events.Error.Error387,FALSE,0);
Error[388].CreateEx(TC_Events.Error.Error388,FALSE,0);
Error[389].CreateEx(TC_Events.Error.Error389,FALSE,0);
Error[390].CreateEx(TC_Events.Error.Error390,FALSE,0);
Error[391].CreateEx(TC_Events.Error.Error391,FALSE,0);
Error[392].CreateEx(TC_Events.Error.Error392,FALSE,0);
Error[393].CreateEx(TC_Events.Error.Error393,FALSE,0);
Error[394].CreateEx(TC_Events.Error.Error394,FALSE,0);
Error[395].CreateEx(TC_Events.Error.Error395,FALSE,0);
Error[396].CreateEx(TC_Events.Error.Error396,FALSE,0);
Error[397].CreateEx(TC_Events.Error.Error397,FALSE,0);
Error[398].CreateEx(TC_Events.Error.Error398,FALSE,0);
Error[399].CreateEx(TC_Events.Error.Error399,FALSE,0);
Error[400].CreateEx(TC_Events.Error.Error400,FALSE,0);
Error[401].CreateEx(TC_Events.Error.Error401,FALSE,0);
Error[402].CreateEx(TC_Events.Error.Error402,FALSE,0);
Error[403].CreateEx(TC_Events.Error.Error403,FALSE,0);
Error[404].CreateEx(TC_Events.Error.Error404,FALSE,0);
Error[405].CreateEx(TC_Events.Error.Error405,FALSE,0);
Error[406].CreateEx(TC_Events.Error.Error406,FALSE,0);
Error[407].CreateEx(TC_Events.Error.Error407,FALSE,0);
Error[408].CreateEx(TC_Events.Error.Error408,FALSE,0);
Error[409].CreateEx(TC_Events.Error.Error409,FALSE,0);
Error[410].CreateEx(TC_Events.Error.Error410,FALSE,0);
Error[411].CreateEx(TC_Events.Error.Error411,FALSE,0);
Error[412].CreateEx(TC_Events.Error.Error412,FALSE,0);
Error[413].CreateEx(TC_Events.Error.Error413,FALSE,0);
Error[414].CreateEx(TC_Events.Error.Error414,FALSE,0);
Error[415].CreateEx(TC_Events.Error.Error415,FALSE,0);
Error[416].CreateEx(TC_Events.Error.Error416,FALSE,0);
Error[417].CreateEx(TC_Events.Error.Error417,FALSE,0);
Error[418].CreateEx(TC_Events.Error.Error418,FALSE,0);
Error[419].CreateEx(TC_Events.Error.Error419,FALSE,0);
Error[420].CreateEx(TC_Events.Error.Error420,FALSE,0);
Error[421].CreateEx(TC_Events.Error.Error421,FALSE,0);
Error[422].CreateEx(TC_Events.Error.Error422,FALSE,0);
Error[423].CreateEx(TC_Events.Error.Error423,FALSE,0);
Error[424].CreateEx(TC_Events.Error.Error424,FALSE,0);
Error[425].CreateEx(TC_Events.Error.Error425,FALSE,0);
Error[426].CreateEx(TC_Events.Error.Error426,FALSE,0);
Error[427].CreateEx(TC_Events.Error.Error427,FALSE,0);
Error[428].CreateEx(TC_Events.Error.Error428,FALSE,0);
Error[429].CreateEx(TC_Events.Error.Error429,FALSE,0);
Error[430].CreateEx(TC_Events.Error.Error430,FALSE,0);
Error[431].CreateEx(TC_Events.Error.Error431,FALSE,0);
Error[432].CreateEx(TC_Events.Error.Error432,FALSE,0);
Error[433].CreateEx(TC_Events.Error.Error433,FALSE,0);
Error[434].CreateEx(TC_Events.Error.Error434,FALSE,0);
Error[435].CreateEx(TC_Events.Error.Error435,FALSE,0);
Error[436].CreateEx(TC_Events.Error.Error436,FALSE,0);
Error[437].CreateEx(TC_Events.Error.Error437,FALSE,0);
Error[438].CreateEx(TC_Events.Error.Error438,FALSE,0);
Error[439].CreateEx(TC_Events.Error.Error439,FALSE,0);
Error[440].CreateEx(TC_Events.Error.Error440,FALSE,0);
Error[441].CreateEx(TC_Events.Error.Error441,FALSE,0);
Error[442].CreateEx(TC_Events.Error.Error442,FALSE,0);
Error[443].CreateEx(TC_Events.Error.Error443,FALSE,0);
Error[444].CreateEx(TC_Events.Error.Error444,FALSE,0);
Error[445].CreateEx(TC_Events.Error.Error445,FALSE,0);
Error[446].CreateEx(TC_Events.Error.Error446,FALSE,0);
Error[447].CreateEx(TC_Events.Error.Error447,FALSE,0);
Error[448].CreateEx(TC_Events.Error.Error448,FALSE,0);
Error[449].CreateEx(TC_Events.Error.Error449,FALSE,0);
Error[450].CreateEx(TC_Events.Error.Error450,FALSE,0);
Error[451].CreateEx(TC_Events.Error.Error451,FALSE,0);
Error[452].CreateEx(TC_Events.Error.Error452,FALSE,0);
Error[453].CreateEx(TC_Events.Error.Error453,FALSE,0);
Error[454].CreateEx(TC_Events.Error.Error454,FALSE,0);
Error[455].CreateEx(TC_Events.Error.Error455,FALSE,0);
Error[456].CreateEx(TC_Events.Error.Error456,FALSE,0);
Error[457].CreateEx(TC_Events.Error.Error457,FALSE,0);
Error[458].CreateEx(TC_Events.Error.Error458,FALSE,0);
Error[459].CreateEx(TC_Events.Error.Error459,FALSE,0);
Error[460].CreateEx(TC_Events.Error.Error460,FALSE,0);
Error[461].CreateEx(TC_Events.Error.Error461,FALSE,0);
Error[462].CreateEx(TC_Events.Error.Error462,FALSE,0);
Error[463].CreateEx(TC_Events.Error.Error463,FALSE,0);
Error[464].CreateEx(TC_Events.Error.Error464,FALSE,0);
Error[465].CreateEx(TC_Events.Error.Error465,FALSE,0);
Error[466].CreateEx(TC_Events.Error.Error466,FALSE,0);
Error[467].CreateEx(TC_Events.Error.Error467,FALSE,0);
Error[468].CreateEx(TC_Events.Error.Error468,FALSE,0);
Error[469].CreateEx(TC_Events.Error.Error469,FALSE,0);
Error[470].CreateEx(TC_Events.Error.Error470,FALSE,0);
Error[471].CreateEx(TC_Events.Error.Error471,FALSE,0);
Error[472].CreateEx(TC_Events.Error.Error472,FALSE,0);
Error[473].CreateEx(TC_Events.Error.Error473,FALSE,0);
Error[474].CreateEx(TC_Events.Error.Error474,FALSE,0);
Error[475].CreateEx(TC_Events.Error.Error475,FALSE,0);
Error[476].CreateEx(TC_Events.Error.Error476,FALSE,0);
Error[477].CreateEx(TC_Events.Error.Error477,FALSE,0);
Error[478].CreateEx(TC_Events.Error.Error478,FALSE,0);
Error[479].CreateEx(TC_Events.Error.Error479,FALSE,0);
Error[480].CreateEx(TC_Events.Error.Error480,FALSE,0);
Error[481].CreateEx(TC_Events.Error.Error481,FALSE,0);
Error[482].CreateEx(TC_Events.Error.Error482,FALSE,0);
Error[483].CreateEx(TC_Events.Error.Error483,FALSE,0);
Error[484].CreateEx(TC_Events.Error.Error484,FALSE,0);
Error[485].CreateEx(TC_Events.Error.Error485,FALSE,0);
Error[486].CreateEx(TC_Events.Error.Error486,FALSE,0);
Error[487].CreateEx(TC_Events.Error.Error487,FALSE,0);
Error[488].CreateEx(TC_Events.Error.Error488,FALSE,0);
Error[489].CreateEx(TC_Events.Error.Error489,FALSE,0);
Error[490].CreateEx(TC_Events.Error.Error490,FALSE,0);
Error[491].CreateEx(TC_Events.Error.Error491,FALSE,0);
Error[492].CreateEx(TC_Events.Error.Error492,FALSE,0);
Error[493].CreateEx(TC_Events.Error.Error493,FALSE,0);
Error[494].CreateEx(TC_Events.Error.Error494,FALSE,0);
Error[495].CreateEx(TC_Events.Error.Error495,FALSE,0);
Error[496].CreateEx(TC_Events.Error.Error496,FALSE,0);
Error[497].CreateEx(TC_Events.Error.Error497,FALSE,0);
Error[498].CreateEx(TC_Events.Error.Error498,FALSE,0);
Error[499].CreateEx(TC_Events.Error.Error499,FALSE,0);
Error[500].CreateEx(TC_Events.Error.Error500,FALSE,0);
Error[501].CreateEx(TC_Events.Error.Error501,FALSE,0);
Error[502].CreateEx(TC_Events.Error.Error502,FALSE,0);
Error[503].CreateEx(TC_Events.Error.Error503,FALSE,0);
Error[504].CreateEx(TC_Events.Error.Error504,FALSE,0);
Error[505].CreateEx(TC_Events.Error.Error505,FALSE,0);
Error[506].CreateEx(TC_Events.Error.Error506,FALSE,0);
Error[507].CreateEx(TC_Events.Error.Error507,FALSE,0);
Error[508].CreateEx(TC_Events.Error.Error508,FALSE,0);
Error[509].CreateEx(TC_Events.Error.Error509,FALSE,0);
Error[510].CreateEx(TC_Events.Error.Error510,FALSE,0);
Error[511].CreateEx(TC_Events.Error.Error511,FALSE,0);
Error[512].CreateEx(TC_Events.Error.Error512,FALSE,0);
Error[513].CreateEx(TC_Events.Error.Error513,FALSE,0);
Error[514].CreateEx(TC_Events.Error.Error514,FALSE,0);
Error[515].CreateEx(TC_Events.Error.Error515,FALSE,0);
Error[516].CreateEx(TC_Events.Error.Error516,FALSE,0);
Error[517].CreateEx(TC_Events.Error.Error517,FALSE,0);
Error[518].CreateEx(TC_Events.Error.Error518,FALSE,0);
Error[519].CreateEx(TC_Events.Error.Error519,FALSE,0);
Error[520].CreateEx(TC_Events.Error.Error520,FALSE,0);
Error[521].CreateEx(TC_Events.Error.Error521,FALSE,0);
Error[522].CreateEx(TC_Events.Error.Error522,FALSE,0);
Error[523].CreateEx(TC_Events.Error.Error523,FALSE,0);
Error[524].CreateEx(TC_Events.Error.Error524,FALSE,0);
Error[525].CreateEx(TC_Events.Error.Error525,FALSE,0);
Error[526].CreateEx(TC_Events.Error.Error526,FALSE,0);
Error[527].CreateEx(TC_Events.Error.Error527,FALSE,0);
Error[528].CreateEx(TC_Events.Error.Error528,FALSE,0);
Error[529].CreateEx(TC_Events.Error.Error529,FALSE,0);
Error[530].CreateEx(TC_Events.Error.Error530,FALSE,0);
Error[531].CreateEx(TC_Events.Error.Error531,FALSE,0);
Error[532].CreateEx(TC_Events.Error.Error532,FALSE,0);
Error[533].CreateEx(TC_Events.Error.Error533,FALSE,0);
Error[534].CreateEx(TC_Events.Error.Error534,FALSE,0);
Error[535].CreateEx(TC_Events.Error.Error535,FALSE,0);
Error[536].CreateEx(TC_Events.Error.Error536,FALSE,0);
Error[537].CreateEx(TC_Events.Error.Error537,FALSE,0);
Error[538].CreateEx(TC_Events.Error.Error538,FALSE,0);
Error[539].CreateEx(TC_Events.Error.Error539,FALSE,0);
Error[540].CreateEx(TC_Events.Error.Error540,FALSE,0);
Error[541].CreateEx(TC_Events.Error.Error541,FALSE,0);
Error[542].CreateEx(TC_Events.Error.Error542,FALSE,0);
Error[543].CreateEx(TC_Events.Error.Error543,FALSE,0);
Error[544].CreateEx(TC_Events.Error.Error544,FALSE,0);
Error[545].CreateEx(TC_Events.Error.Error545,FALSE,0);
Error[546].CreateEx(TC_Events.Error.Error546,FALSE,0);
Error[547].CreateEx(TC_Events.Error.Error547,FALSE,0);
Error[548].CreateEx(TC_Events.Error.Error548,FALSE,0);
Error[549].CreateEx(TC_Events.Error.Error549,FALSE,0);
Error[550].CreateEx(TC_Events.Error.Error550,FALSE,0);
Error[551].CreateEx(TC_Events.Error.Error551,FALSE,0);
Error[552].CreateEx(TC_Events.Error.Error552,FALSE,0);
Error[553].CreateEx(TC_Events.Error.Error553,FALSE,0);
Error[554].CreateEx(TC_Events.Error.Error554,FALSE,0);
Error[555].CreateEx(TC_Events.Error.Error555,FALSE,0);
Error[556].CreateEx(TC_Events.Error.Error556,FALSE,0);
Error[557].CreateEx(TC_Events.Error.Error557,FALSE,0);
Error[558].CreateEx(TC_Events.Error.Error558,FALSE,0);
Error[559].CreateEx(TC_Events.Error.Error559,FALSE,0);
Error[560].CreateEx(TC_Events.Error.Error560,FALSE,0);
Error[561].CreateEx(TC_Events.Error.Error561,FALSE,0);
Error[562].CreateEx(TC_Events.Error.Error562,FALSE,0);
Error[563].CreateEx(TC_Events.Error.Error563,FALSE,0);
Error[564].CreateEx(TC_Events.Error.Error564,FALSE,0);
Error[565].CreateEx(TC_Events.Error.Error565,FALSE,0);
Error[566].CreateEx(TC_Events.Error.Error566,FALSE,0);
Error[567].CreateEx(TC_Events.Error.Error567,FALSE,0);
Error[568].CreateEx(TC_Events.Error.Error568,FALSE,0);
Error[569].CreateEx(TC_Events.Error.Error569,FALSE,0);
Error[570].CreateEx(TC_Events.Error.Error570,FALSE,0);
Error[571].CreateEx(TC_Events.Error.Error571,FALSE,0);
Error[572].CreateEx(TC_Events.Error.Error572,FALSE,0);
Error[573].CreateEx(TC_Events.Error.Error573,FALSE,0);
Error[574].CreateEx(TC_Events.Error.Error574,FALSE,0);
Error[575].CreateEx(TC_Events.Error.Error575,FALSE,0);
Error[576].CreateEx(TC_Events.Error.Error576,FALSE,0);
Error[577].CreateEx(TC_Events.Error.Error577,FALSE,0);
Error[578].CreateEx(TC_Events.Error.Error578,FALSE,0);
Error[579].CreateEx(TC_Events.Error.Error579,FALSE,0);
Error[580].CreateEx(TC_Events.Error.Error580,FALSE,0);
Error[581].CreateEx(TC_Events.Error.Error581,FALSE,0);
Error[582].CreateEx(TC_Events.Error.Error582,FALSE,0);
Error[583].CreateEx(TC_Events.Error.Error583,FALSE,0);
Error[584].CreateEx(TC_Events.Error.Error584,FALSE,0);
Error[585].CreateEx(TC_Events.Error.Error585,FALSE,0);
Error[586].CreateEx(TC_Events.Error.Error586,FALSE,0);
Error[587].CreateEx(TC_Events.Error.Error587,FALSE,0);
Error[588].CreateEx(TC_Events.Error.Error588,FALSE,0);
Error[589].CreateEx(TC_Events.Error.Error589,FALSE,0);
Error[590].CreateEx(TC_Events.Error.Error590,FALSE,0);
Error[591].CreateEx(TC_Events.Error.Error591,FALSE,0);
Error[592].CreateEx(TC_Events.Error.Error592,FALSE,0);
Error[593].CreateEx(TC_Events.Error.Error593,FALSE,0);
Error[594].CreateEx(TC_Events.Error.Error594,FALSE,0);
Error[595].CreateEx(TC_Events.Error.Error595,FALSE,0);
Error[596].CreateEx(TC_Events.Error.Error596,FALSE,0);
Error[597].CreateEx(TC_Events.Error.Error597,FALSE,0);
Error[598].CreateEx(TC_Events.Error.Error598,FALSE,0);
Error[599].CreateEx(TC_Events.Error.Error599,FALSE,0);
Error[600].CreateEx(TC_Events.Error.Error600,FALSE,0);
Error[601].CreateEx(TC_Events.Error.Error601,FALSE,0);
Error[602].CreateEx(TC_Events.Error.Error602,FALSE,0);
Error[603].CreateEx(TC_Events.Error.Error603,FALSE,0);
Error[604].CreateEx(TC_Events.Error.Error604,FALSE,0);
Error[605].CreateEx(TC_Events.Error.Error605,FALSE,0);
Error[606].CreateEx(TC_Events.Error.Error606,FALSE,0);
Error[607].CreateEx(TC_Events.Error.Error607,FALSE,0);
Error[608].CreateEx(TC_Events.Error.Error608,FALSE,0);
Error[609].CreateEx(TC_Events.Error.Error609,FALSE,0);
Error[610].CreateEx(TC_Events.Error.Error610,FALSE,0);
Error[611].CreateEx(TC_Events.Error.Error611,FALSE,0);
Error[612].CreateEx(TC_Events.Error.Error612,FALSE,0);
Error[613].CreateEx(TC_Events.Error.Error613,FALSE,0);
Error[614].CreateEx(TC_Events.Error.Error614,FALSE,0);
Error[615].CreateEx(TC_Events.Error.Error615,FALSE,0);
Error[616].CreateEx(TC_Events.Error.Error616,FALSE,0);
Error[617].CreateEx(TC_Events.Error.Error617,FALSE,0);
Error[618].CreateEx(TC_Events.Error.Error618,FALSE,0);
Error[619].CreateEx(TC_Events.Error.Error619,FALSE,0);
Error[620].CreateEx(TC_Events.Error.Error620,FALSE,0);
Error[621].CreateEx(TC_Events.Error.Error621,FALSE,0);
Error[622].CreateEx(TC_Events.Error.Error622,FALSE,0);
Error[623].CreateEx(TC_Events.Error.Error623,FALSE,0);
Error[624].CreateEx(TC_Events.Error.Error624,FALSE,0);
Error[625].CreateEx(TC_Events.Error.Error625,FALSE,0);
Error[626].CreateEx(TC_Events.Error.Error626,FALSE,0);
Error[627].CreateEx(TC_Events.Error.Error627,FALSE,0);
Error[628].CreateEx(TC_Events.Error.Error628,FALSE,0);
Error[629].CreateEx(TC_Events.Error.Error629,FALSE,0);
Error[630].CreateEx(TC_Events.Error.Error630,FALSE,0);
Error[631].CreateEx(TC_Events.Error.Error631,FALSE,0);
Error[632].CreateEx(TC_Events.Error.Error632,FALSE,0);
Error[633].CreateEx(TC_Events.Error.Error633,FALSE,0);
Error[634].CreateEx(TC_Events.Error.Error634,FALSE,0);
Error[635].CreateEx(TC_Events.Error.Error635,FALSE,0);
Error[636].CreateEx(TC_Events.Error.Error636,FALSE,0);
Error[637].CreateEx(TC_Events.Error.Error637,FALSE,0);
Error[638].CreateEx(TC_Events.Error.Error638,FALSE,0);
Error[639].CreateEx(TC_Events.Error.Error639,FALSE,0);
Error[640].CreateEx(TC_Events.Error.Error640,FALSE,0);
Error[641].CreateEx(TC_Events.Error.Error641,FALSE,0);
Error[642].CreateEx(TC_Events.Error.Error642,FALSE,0);
Error[643].CreateEx(TC_Events.Error.Error643,FALSE,0);
Error[644].CreateEx(TC_Events.Error.Error644,FALSE,0);
Error[645].CreateEx(TC_Events.Error.Error645,FALSE,0);
Error[646].CreateEx(TC_Events.Error.Error646,FALSE,0);
Error[647].CreateEx(TC_Events.Error.Error647,FALSE,0);
Error[648].CreateEx(TC_Events.Error.Error648,FALSE,0);
Error[649].CreateEx(TC_Events.Error.Error649,FALSE,0);
Error[650].CreateEx(TC_Events.Error.Error650,FALSE,0);
Error[651].CreateEx(TC_Events.Error.Error651,FALSE,0);
Error[652].CreateEx(TC_Events.Error.Error652,FALSE,0);
Error[653].CreateEx(TC_Events.Error.Error653,FALSE,0);
Error[654].CreateEx(TC_Events.Error.Error654,FALSE,0);
Error[655].CreateEx(TC_Events.Error.Error655,FALSE,0);
Error[656].CreateEx(TC_Events.Error.Error656,FALSE,0);
Error[657].CreateEx(TC_Events.Error.Error657,FALSE,0);
Error[658].CreateEx(TC_Events.Error.Error658,FALSE,0);
Error[659].CreateEx(TC_Events.Error.Error659,FALSE,0);
Error[660].CreateEx(TC_Events.Error.Error660,FALSE,0);
Error[661].CreateEx(TC_Events.Error.Error661,FALSE,0);
Error[662].CreateEx(TC_Events.Error.Error662,FALSE,0);
Error[663].CreateEx(TC_Events.Error.Error663,FALSE,0);
Error[664].CreateEx(TC_Events.Error.Error664,FALSE,0);
Error[665].CreateEx(TC_Events.Error.Error665,FALSE,0);
Error[666].CreateEx(TC_Events.Error.Error666,FALSE,0);
Error[667].CreateEx(TC_Events.Error.Error667,FALSE,0);
Error[668].CreateEx(TC_Events.Error.Error668,FALSE,0);
Error[669].CreateEx(TC_Events.Error.Error669,FALSE,0);
Error[670].CreateEx(TC_Events.Error.Error670,FALSE,0);
Error[671].CreateEx(TC_Events.Error.Error671,FALSE,0);
Error[672].CreateEx(TC_Events.Error.Error672,FALSE,0);
Error[673].CreateEx(TC_Events.Error.Error673,FALSE,0);
Error[674].CreateEx(TC_Events.Error.Error674,FALSE,0);
Error[675].CreateEx(TC_Events.Error.Error675,FALSE,0);
Error[676].CreateEx(TC_Events.Error.Error676,FALSE,0);
Error[677].CreateEx(TC_Events.Error.Error677,FALSE,0);
Error[678].CreateEx(TC_Events.Error.Error678,FALSE,0);
Error[679].CreateEx(TC_Events.Error.Error679,FALSE,0);
Error[680].CreateEx(TC_Events.Error.Error680,FALSE,0);
Error[681].CreateEx(TC_Events.Error.Error681,FALSE,0);
Error[682].CreateEx(TC_Events.Error.Error682,FALSE,0);
Error[683].CreateEx(TC_Events.Error.Error683,FALSE,0);
Error[684].CreateEx(TC_Events.Error.Error684,FALSE,0);
Error[685].CreateEx(TC_Events.Error.Error685,FALSE,0);
Error[686].CreateEx(TC_Events.Error.Error686,FALSE,0);
Error[687].CreateEx(TC_Events.Error.Error687,FALSE,0);
Error[688].CreateEx(TC_Events.Error.Error688,FALSE,0);
Error[689].CreateEx(TC_Events.Error.Error689,FALSE,0);
Error[690].CreateEx(TC_Events.Error.Error690,FALSE,0);
Error[691].CreateEx(TC_Events.Error.Error691,FALSE,0);
Error[692].CreateEx(TC_Events.Error.Error692,FALSE,0);
Error[693].CreateEx(TC_Events.Error.Error693,FALSE,0);
Error[694].CreateEx(TC_Events.Error.Error694,FALSE,0);
Error[695].CreateEx(TC_Events.Error.Error695,FALSE,0);
Error[696].CreateEx(TC_Events.Error.Error696,FALSE,0);
Error[697].CreateEx(TC_Events.Error.Error697,FALSE,0);
Error[698].CreateEx(TC_Events.Error.Error698,FALSE,0);
Error[699].CreateEx(TC_Events.Error.Error699,FALSE,0);
Error[700].CreateEx(TC_Events.Error.Error700,FALSE,0);
Error[701].CreateEx(TC_Events.Error.Error701,FALSE,0);
Error[702].CreateEx(TC_Events.Error.Error702,FALSE,0);
Error[703].CreateEx(TC_Events.Error.Error703,FALSE,0);
Error[704].CreateEx(TC_Events.Error.Error704,FALSE,0);
Error[705].CreateEx(TC_Events.Error.Error705,FALSE,0);
Error[706].CreateEx(TC_Events.Error.Error706,FALSE,0);
Error[707].CreateEx(TC_Events.Error.Error707,FALSE,0);
Error[708].CreateEx(TC_Events.Error.Error708,FALSE,0);
Error[709].CreateEx(TC_Events.Error.Error709,FALSE,0);
Error[710].CreateEx(TC_Events.Error.Error710,FALSE,0);
Error[711].CreateEx(TC_Events.Error.Error711,FALSE,0);
Error[712].CreateEx(TC_Events.Error.Error712,FALSE,0);
Error[713].CreateEx(TC_Events.Error.Error713,FALSE,0);
Error[714].CreateEx(TC_Events.Error.Error714,FALSE,0);
Error[715].CreateEx(TC_Events.Error.Error715,FALSE,0);
Error[716].CreateEx(TC_Events.Error.Error716,FALSE,0);
Error[717].CreateEx(TC_Events.Error.Error717,FALSE,0);
Error[718].CreateEx(TC_Events.Error.Error718,FALSE,0);
Error[719].CreateEx(TC_Events.Error.Error719,FALSE,0);
Error[720].CreateEx(TC_Events.Error.Error720,FALSE,0);
Error[721].CreateEx(TC_Events.Error.Error721,FALSE,0);
Error[722].CreateEx(TC_Events.Error.Error722,FALSE,0);
Error[723].CreateEx(TC_Events.Error.Error723,FALSE,0);
Error[724].CreateEx(TC_Events.Error.Error724,FALSE,0);
Error[725].CreateEx(TC_Events.Error.Error725,FALSE,0);
Error[726].CreateEx(TC_Events.Error.Error726,FALSE,0);
Error[727].CreateEx(TC_Events.Error.Error727,FALSE,0);
Error[728].CreateEx(TC_Events.Error.Error728,FALSE,0);
Error[729].CreateEx(TC_Events.Error.Error729,FALSE,0);
Error[730].CreateEx(TC_Events.Error.Error730,FALSE,0);
Error[731].CreateEx(TC_Events.Error.Error731,FALSE,0);
Error[732].CreateEx(TC_Events.Error.Error732,FALSE,0);
Error[733].CreateEx(TC_Events.Error.Error733,FALSE,0);
Error[734].CreateEx(TC_Events.Error.Error734,FALSE,0);
Error[735].CreateEx(TC_Events.Error.Error735,FALSE,0);
Error[736].CreateEx(TC_Events.Error.Error736,FALSE,0);
Error[737].CreateEx(TC_Events.Error.Error737,FALSE,0);
Error[738].CreateEx(TC_Events.Error.Error738,FALSE,0);
Error[739].CreateEx(TC_Events.Error.Error739,FALSE,0);
Error[740].CreateEx(TC_Events.Error.Error740,FALSE,0);
Error[741].CreateEx(TC_Events.Error.Error741,FALSE,0);
Error[742].CreateEx(TC_Events.Error.Error742,FALSE,0);
Error[743].CreateEx(TC_Events.Error.Error743,FALSE,0);
Error[744].CreateEx(TC_Events.Error.Error744,FALSE,0);
Error[745].CreateEx(TC_Events.Error.Error745,FALSE,0);
Error[746].CreateEx(TC_Events.Error.Error746,FALSE,0);
Error[747].CreateEx(TC_Events.Error.Error747,FALSE,0);
Error[748].CreateEx(TC_Events.Error.Error748,FALSE,0);
Error[749].CreateEx(TC_Events.Error.Error749,FALSE,0);
Error[750].CreateEx(TC_Events.Error.Error750,FALSE,0);
Error[751].CreateEx(TC_Events.Error.Error751,FALSE,0);
Error[752].CreateEx(TC_Events.Error.Error752,FALSE,0);
Error[753].CreateEx(TC_Events.Error.Error753,FALSE,0);
Error[754].CreateEx(TC_Events.Error.Error754,FALSE,0);
Error[755].CreateEx(TC_Events.Error.Error755,FALSE,0);
Error[756].CreateEx(TC_Events.Error.Error756,FALSE,0);
Error[757].CreateEx(TC_Events.Error.Error757,FALSE,0);
Error[758].CreateEx(TC_Events.Error.Error758,FALSE,0);
Error[759].CreateEx(TC_Events.Error.Error759,FALSE,0);
Error[760].CreateEx(TC_Events.Error.Error760,FALSE,0);
Error[761].CreateEx(TC_Events.Error.Error761,FALSE,0);
Error[762].CreateEx(TC_Events.Error.Error762,FALSE,0);
Error[763].CreateEx(TC_Events.Error.Error763,FALSE,0);
Error[764].CreateEx(TC_Events.Error.Error764,FALSE,0);
Error[765].CreateEx(TC_Events.Error.Error765,FALSE,0);
Error[766].CreateEx(TC_Events.Error.Error766,FALSE,0);
Error[767].CreateEx(TC_Events.Error.Error767,FALSE,0);
Error[768].CreateEx(TC_Events.Error.Error768,FALSE,0);
Error[769].CreateEx(TC_Events.Error.Error769,FALSE,0);
Error[770].CreateEx(TC_Events.Error.Error770,FALSE,0);
Error[771].CreateEx(TC_Events.Error.Error771,FALSE,0);
Error[772].CreateEx(TC_Events.Error.Error772,FALSE,0);
Error[773].CreateEx(TC_Events.Error.Error773,FALSE,0);
Error[774].CreateEx(TC_Events.Error.Error774,FALSE,0);
Error[775].CreateEx(TC_Events.Error.Error775,FALSE,0);
Error[776].CreateEx(TC_Events.Error.Error776,FALSE,0);
Error[777].CreateEx(TC_Events.Error.Error777,FALSE,0);
Error[778].CreateEx(TC_Events.Error.Error778,FALSE,0);
Error[779].CreateEx(TC_Events.Error.Error779,FALSE,0);
Error[780].CreateEx(TC_Events.Error.Error780,FALSE,0);
Error[781].CreateEx(TC_Events.Error.Error781,FALSE,0);
Error[782].CreateEx(TC_Events.Error.Error782,FALSE,0);
Error[783].CreateEx(TC_Events.Error.Error783,FALSE,0);
Error[784].CreateEx(TC_Events.Error.Error784,FALSE,0);
Error[785].CreateEx(TC_Events.Error.Error785,FALSE,0);
Error[786].CreateEx(TC_Events.Error.Error786,FALSE,0);
Error[787].CreateEx(TC_Events.Error.Error787,FALSE,0);
Error[788].CreateEx(TC_Events.Error.Error788,FALSE,0);
Error[789].CreateEx(TC_Events.Error.Error789,FALSE,0);
Error[790].CreateEx(TC_Events.Error.Error790,FALSE,0);
Error[791].CreateEx(TC_Events.Error.Error791,FALSE,0);
Error[792].CreateEx(TC_Events.Error.Error792,FALSE,0);
Error[793].CreateEx(TC_Events.Error.Error793,FALSE,0);
Error[794].CreateEx(TC_Events.Error.Error794,FALSE,0);
Error[795].CreateEx(TC_Events.Error.Error795,FALSE,0);
Error[796].CreateEx(TC_Events.Error.Error796,FALSE,0);
Error[797].CreateEx(TC_Events.Error.Error797,FALSE,0);
Error[798].CreateEx(TC_Events.Error.Error798,FALSE,0);
Error[799].CreateEx(TC_Events.Error.Error799,FALSE,0);
Error[800].CreateEx(TC_Events.Error.Error800,FALSE,0);
Error[801].CreateEx(TC_Events.Error.Error801,FALSE,0);
Error[802].CreateEx(TC_Events.Error.Error802,FALSE,0);
Error[803].CreateEx(TC_Events.Error.Error803,FALSE,0);
Error[804].CreateEx(TC_Events.Error.Error804,FALSE,0);
Error[805].CreateEx(TC_Events.Error.Error805,FALSE,0);
Error[806].CreateEx(TC_Events.Error.Error806,FALSE,0);
Error[807].CreateEx(TC_Events.Error.Error807,FALSE,0);
Error[808].CreateEx(TC_Events.Error.Error808,FALSE,0);
Error[809].CreateEx(TC_Events.Error.Error809,FALSE,0);
Error[810].CreateEx(TC_Events.Error.Error810,FALSE,0);
Error[811].CreateEx(TC_Events.Error.Error811,FALSE,0);
Error[812].CreateEx(TC_Events.Error.Error812,FALSE,0);
Error[813].CreateEx(TC_Events.Error.Error813,FALSE,0);
Error[814].CreateEx(TC_Events.Error.Error814,FALSE,0);
Error[815].CreateEx(TC_Events.Error.Error815,FALSE,0);
Error[816].CreateEx(TC_Events.Error.Error816,FALSE,0);
Error[817].CreateEx(TC_Events.Error.Error817,FALSE,0);
Error[818].CreateEx(TC_Events.Error.Error818,FALSE,0);
Error[819].CreateEx(TC_Events.Error.Error819,FALSE,0);
Error[820].CreateEx(TC_Events.Error.Error820,FALSE,0);
Error[821].CreateEx(TC_Events.Error.Error821,FALSE,0);
Error[822].CreateEx(TC_Events.Error.Error822,FALSE,0);
Error[823].CreateEx(TC_Events.Error.Error823,FALSE,0);
Error[824].CreateEx(TC_Events.Error.Error824,FALSE,0);
Error[825].CreateEx(TC_Events.Error.Error825,FALSE,0);
Error[826].CreateEx(TC_Events.Error.Error826,FALSE,0);
Error[827].CreateEx(TC_Events.Error.Error827,FALSE,0);
Error[828].CreateEx(TC_Events.Error.Error828,FALSE,0);
Error[829].CreateEx(TC_Events.Error.Error829,FALSE,0);
Error[830].CreateEx(TC_Events.Error.Error830,FALSE,0);
Error[831].CreateEx(TC_Events.Error.Error831,FALSE,0);
Error[832].CreateEx(TC_Events.Error.Error832,FALSE,0);
Error[833].CreateEx(TC_Events.Error.Error833,FALSE,0);
Error[834].CreateEx(TC_Events.Error.Error834,FALSE,0);
Error[835].CreateEx(TC_Events.Error.Error835,FALSE,0);
Error[836].CreateEx(TC_Events.Error.Error836,FALSE,0);
Error[837].CreateEx(TC_Events.Error.Error837,FALSE,0);
Error[838].CreateEx(TC_Events.Error.Error838,FALSE,0);
Error[839].CreateEx(TC_Events.Error.Error839,FALSE,0);
Error[840].CreateEx(TC_Events.Error.Error840,FALSE,0);
Error[841].CreateEx(TC_Events.Error.Error841,FALSE,0);
Error[842].CreateEx(TC_Events.Error.Error842,FALSE,0);
Error[843].CreateEx(TC_Events.Error.Error843,FALSE,0);
Error[844].CreateEx(TC_Events.Error.Error844,FALSE,0);
Error[845].CreateEx(TC_Events.Error.Error845,FALSE,0);
Error[846].CreateEx(TC_Events.Error.Error846,FALSE,0);
Error[847].CreateEx(TC_Events.Error.Error847,FALSE,0);
Error[848].CreateEx(TC_Events.Error.Error848,FALSE,0);
Error[849].CreateEx(TC_Events.Error.Error849,FALSE,0);
Error[850].CreateEx(TC_Events.Error.Error850,FALSE,0);
Error[851].CreateEx(TC_Events.Error.Error851,FALSE,0);
Error[852].CreateEx(TC_Events.Error.Error852,FALSE,0);
Error[853].CreateEx(TC_Events.Error.Error853,FALSE,0);
Error[854].CreateEx(TC_Events.Error.Error854,FALSE,0);
Error[855].CreateEx(TC_Events.Error.Error855,FALSE,0);
Error[856].CreateEx(TC_Events.Error.Error856,FALSE,0);
Error[857].CreateEx(TC_Events.Error.Error857,FALSE,0);
Error[858].CreateEx(TC_Events.Error.Error858,FALSE,0);
Error[859].CreateEx(TC_Events.Error.Error859,FALSE,0);
Error[860].CreateEx(TC_Events.Error.Error860,FALSE,0);
Error[861].CreateEx(TC_Events.Error.Error861,FALSE,0);
Error[862].CreateEx(TC_Events.Error.Error862,FALSE,0);
Error[863].CreateEx(TC_Events.Error.Error863,FALSE,0);
Error[864].CreateEx(TC_Events.Error.Error864,FALSE,0);
Error[865].CreateEx(TC_Events.Error.Error865,FALSE,0);
Error[866].CreateEx(TC_Events.Error.Error866,FALSE,0);
Error[867].CreateEx(TC_Events.Error.Error867,FALSE,0);
Error[868].CreateEx(TC_Events.Error.Error868,FALSE,0);
Error[869].CreateEx(TC_Events.Error.Error869,FALSE,0);
Error[870].CreateEx(TC_Events.Error.Error870,FALSE,0);
Error[871].CreateEx(TC_Events.Error.Error871,FALSE,0);
Error[872].CreateEx(TC_Events.Error.Error872,FALSE,0);
Error[873].CreateEx(TC_Events.Error.Error873,FALSE,0);
Error[874].CreateEx(TC_Events.Error.Error874,FALSE,0);
Error[875].CreateEx(TC_Events.Error.Error875,FALSE,0);
Error[876].CreateEx(TC_Events.Error.Error876,FALSE,0);
Error[877].CreateEx(TC_Events.Error.Error877,FALSE,0);
Error[878].CreateEx(TC_Events.Error.Error878,FALSE,0);
Error[879].CreateEx(TC_Events.Error.Error879,FALSE,0);
Error[880].CreateEx(TC_Events.Error.Error880,FALSE,0);
Error[881].CreateEx(TC_Events.Error.Error881,FALSE,0);
Error[882].CreateEx(TC_Events.Error.Error882,FALSE,0);
Error[883].CreateEx(TC_Events.Error.Error883,FALSE,0);
Error[884].CreateEx(TC_Events.Error.Error884,FALSE,0);
Error[885].CreateEx(TC_Events.Error.Error885,FALSE,0);
Error[886].CreateEx(TC_Events.Error.Error886,FALSE,0);
Error[887].CreateEx(TC_Events.Error.Error887,FALSE,0);
Error[888].CreateEx(TC_Events.Error.Error888,FALSE,0);
Error[889].CreateEx(TC_Events.Error.Error889,FALSE,0);
Error[890].CreateEx(TC_Events.Error.Error890,FALSE,0);
Error[891].CreateEx(TC_Events.Error.Error891,FALSE,0);
Error[892].CreateEx(TC_Events.Error.Error892,FALSE,0);
Error[893].CreateEx(TC_Events.Error.Error893,FALSE,0);
Error[894].CreateEx(TC_Events.Error.Error894,FALSE,0);
Error[895].CreateEx(TC_Events.Error.Error895,FALSE,0);
Error[896].CreateEx(TC_Events.Error.Error896,FALSE,0);
Error[897].CreateEx(TC_Events.Error.Error897,FALSE,0);
Error[898].CreateEx(TC_Events.Error.Error898,FALSE,0);
Error[899].CreateEx(TC_Events.Error.Error899,FALSE,0);
Error[900].CreateEx(TC_Events.Error.Error900,FALSE,0);
Error[901].CreateEx(TC_Events.Error.Error901,FALSE,0);
Error[902].CreateEx(TC_Events.Error.Error902,FALSE,0);
Error[903].CreateEx(TC_Events.Error.Error903,FALSE,0);
Error[904].CreateEx(TC_Events.Error.Error904,FALSE,0);
Error[905].CreateEx(TC_Events.Error.Error905,FALSE,0);
Error[906].CreateEx(TC_Events.Error.Error906,FALSE,0);
Error[907].CreateEx(TC_Events.Error.Error907,FALSE,0);
Error[908].CreateEx(TC_Events.Error.Error908,FALSE,0);
Error[909].CreateEx(TC_Events.Error.Error909,FALSE,0);
Error[910].CreateEx(TC_Events.Error.Error910,FALSE,0);
Error[911].CreateEx(TC_Events.Error.Error911,FALSE,0);
Error[912].CreateEx(TC_Events.Error.Error912,FALSE,0);
Error[913].CreateEx(TC_Events.Error.Error913,FALSE,0);
Error[914].CreateEx(TC_Events.Error.Error914,FALSE,0);
Error[915].CreateEx(TC_Events.Error.Error915,FALSE,0);
Error[916].CreateEx(TC_Events.Error.Error916,FALSE,0);
Error[917].CreateEx(TC_Events.Error.Error917,FALSE,0);
Error[918].CreateEx(TC_Events.Error.Error918,FALSE,0);
Error[919].CreateEx(TC_Events.Error.Error919,FALSE,0);
Error[920].CreateEx(TC_Events.Error.Error920,FALSE,0);
Error[921].CreateEx(TC_Events.Error.Error921,FALSE,0);
Error[922].CreateEx(TC_Events.Error.Error922,FALSE,0);
Error[923].CreateEx(TC_Events.Error.Error923,FALSE,0);
Error[924].CreateEx(TC_Events.Error.Error924,FALSE,0);
Error[925].CreateEx(TC_Events.Error.Error925,FALSE,0);
Error[926].CreateEx(TC_Events.Error.Error926,FALSE,0);
Error[927].CreateEx(TC_Events.Error.Error927,FALSE,0);
Error[928].CreateEx(TC_Events.Error.Error928,FALSE,0);
Error[929].CreateEx(TC_Events.Error.Error929,FALSE,0);
Error[930].CreateEx(TC_Events.Error.Error930,FALSE,0);
Error[931].CreateEx(TC_Events.Error.Error931,FALSE,0);
Error[932].CreateEx(TC_Events.Error.Error932,FALSE,0);
Error[933].CreateEx(TC_Events.Error.Error933,FALSE,0);
Error[934].CreateEx(TC_Events.Error.Error934,FALSE,0);
Error[935].CreateEx(TC_Events.Error.Error935,FALSE,0);
Error[936].CreateEx(TC_Events.Error.Error936,FALSE,0);
Error[937].CreateEx(TC_Events.Error.Error937,FALSE,0);
Error[938].CreateEx(TC_Events.Error.Error938,FALSE,0);
Error[939].CreateEx(TC_Events.Error.Error939,FALSE,0);
Error[940].CreateEx(TC_Events.Error.Error940,FALSE,0);
Error[941].CreateEx(TC_Events.Error.Error941,FALSE,0);
Error[942].CreateEx(TC_Events.Error.Error942,FALSE,0);
Error[943].CreateEx(TC_Events.Error.Error943,FALSE,0);
Error[944].CreateEx(TC_Events.Error.Error944,FALSE,0);
Error[945].CreateEx(TC_Events.Error.Error945,FALSE,0);
Error[946].CreateEx(TC_Events.Error.Error946,FALSE,0);
Error[947].CreateEx(TC_Events.Error.Error947,FALSE,0);
Error[948].CreateEx(TC_Events.Error.Error948,FALSE,0);
Error[949].CreateEx(TC_Events.Error.Error949,FALSE,0);
Error[950].CreateEx(TC_Events.Error.Error950,FALSE,0);
Error[951].CreateEx(TC_Events.Error.Error951,FALSE,0);
Error[952].CreateEx(TC_Events.Error.Error952,FALSE,0);
Error[953].CreateEx(TC_Events.Error.Error953,FALSE,0);
Error[954].CreateEx(TC_Events.Error.Error954,FALSE,0);
Error[955].CreateEx(TC_Events.Error.Error955,FALSE,0);
Error[956].CreateEx(TC_Events.Error.Error956,FALSE,0);
Error[957].CreateEx(TC_Events.Error.Error957,FALSE,0);
Error[958].CreateEx(TC_Events.Error.Error958,FALSE,0);
Error[959].CreateEx(TC_Events.Error.Error959,FALSE,0);
Error[960].CreateEx(TC_Events.Error.Error960,FALSE,0);
Error[961].CreateEx(TC_Events.Error.Error961,FALSE,0);
Error[962].CreateEx(TC_Events.Error.Error962,FALSE,0);
Error[963].CreateEx(TC_Events.Error.Error963,FALSE,0);
Error[964].CreateEx(TC_Events.Error.Error964,FALSE,0);
Error[965].CreateEx(TC_Events.Error.Error965,FALSE,0);
Error[966].CreateEx(TC_Events.Error.Error966,FALSE,0);
Error[967].CreateEx(TC_Events.Error.Error967,FALSE,0);
Error[968].CreateEx(TC_Events.Error.Error968,FALSE,0);
Error[969].CreateEx(TC_Events.Error.Error969,FALSE,0);
Error[970].CreateEx(TC_Events.Error.Error970,FALSE,0);
Error[971].CreateEx(TC_Events.Error.Error971,FALSE,0);
Error[972].CreateEx(TC_Events.Error.Error972,FALSE,0);
Error[973].CreateEx(TC_Events.Error.Error973,FALSE,0);
Error[974].CreateEx(TC_Events.Error.Error974,FALSE,0);
Error[975].CreateEx(TC_Events.Error.Error975,FALSE,0);
Error[976].CreateEx(TC_Events.Error.Error976,FALSE,0);
Error[977].CreateEx(TC_Events.Error.Error977,FALSE,0);
Error[978].CreateEx(TC_Events.Error.Error978,FALSE,0);
Error[979].CreateEx(TC_Events.Error.Error979,FALSE,0);
Error[980].CreateEx(TC_Events.Error.Error980,FALSE,0);
Error[981].CreateEx(TC_Events.Error.Error981,FALSE,0);
Error[982].CreateEx(TC_Events.Error.Error982,FALSE,0);
Error[983].CreateEx(TC_Events.Error.Error983,FALSE,0);
Error[984].CreateEx(TC_Events.Error.Error984,FALSE,0);
Error[985].CreateEx(TC_Events.Error.Error985,FALSE,0);
Error[986].CreateEx(TC_Events.Error.Error986,FALSE,0);
Error[987].CreateEx(TC_Events.Error.Error987,FALSE,0);
Error[988].CreateEx(TC_Events.Error.Error988,FALSE,0);
Error[989].CreateEx(TC_Events.Error.Error989,FALSE,0);
Error[990].CreateEx(TC_Events.Error.Error990,FALSE,0);
Error[991].CreateEx(TC_Events.Error.Error991,FALSE,0);
Error[992].CreateEx(TC_Events.Error.Error992,FALSE,0);
Error[993].CreateEx(TC_Events.Error.Error993,FALSE,0);
Error[994].CreateEx(TC_Events.Error.Error994,FALSE,0);
Error[995].CreateEx(TC_Events.Error.Error995,FALSE,0);
Error[996].CreateEx(TC_Events.Error.Error996,FALSE,0);
Error[997].CreateEx(TC_Events.Error.Error997,FALSE,0);
Error[998].CreateEx(TC_Events.Error.Error998,FALSE,0);
Error[999].CreateEx(TC_Events.Error.Error999,FALSE,0);
Error[1000].CreateEx(TC_Events.Error.Error1000,FALSE,0);
Error[1001].CreateEx(TC_Events.Error.Error1001,FALSE,0);
Error[1002].CreateEx(TC_Events.Error.Error1002,FALSE,0);
Error[1003].CreateEx(TC_Events.Error.Error1003,FALSE,0);
Error[1004].CreateEx(TC_Events.Error.Error1004,FALSE,0);
Error[1005].CreateEx(TC_Events.Error.Error1005,FALSE,0);
Error[1006].CreateEx(TC_Events.Error.Error1006,FALSE,0);
Error[1007].CreateEx(TC_Events.Error.Error1007,FALSE,0);
Error[1008].CreateEx(TC_Events.Error.Error1008,FALSE,0);
Error[1009].CreateEx(TC_Events.Error.Error1009,FALSE,0);
Error[1010].CreateEx(TC_Events.Error.Error1010,FALSE,0);
Error[1011].CreateEx(TC_Events.Error.Error1011,FALSE,0);
Error[1012].CreateEx(TC_Events.Error.Error1012,FALSE,0);
Error[1013].CreateEx(TC_Events.Error.Error1013,FALSE,0);
Error[1014].CreateEx(TC_Events.Error.Error1014,FALSE,0);
Error[1015].CreateEx(TC_Events.Error.Error1015,FALSE,0);
Error[1016].CreateEx(TC_Events.Error.Error1016,FALSE,0);
Error[1017].CreateEx(TC_Events.Error.Error1017,FALSE,0);
Error[1018].CreateEx(TC_Events.Error.Error1018,FALSE,0);
Error[1019].CreateEx(TC_Events.Error.Error1019,FALSE,0);
Error[1020].CreateEx(TC_Events.Error.Error1020,FALSE,0);
Error[1021].CreateEx(TC_Events.Error.Error1021,FALSE,0);
Error[1022].CreateEx(TC_Events.Error.Error1022,FALSE,0);
Error[1023].CreateEx(TC_Events.Error.Error1023,FALSE,0);
Error[1024].CreateEx(TC_Events.Error.Error1024,FALSE,0);
Error[1025].CreateEx(TC_Events.Error.Error1025,FALSE,0);
Error[1026].CreateEx(TC_Events.Error.Error1026,FALSE,0);
Error[1027].CreateEx(TC_Events.Error.Error1027,FALSE,0);
Error[1028].CreateEx(TC_Events.Error.Error1028,FALSE,0);
Error[1029].CreateEx(TC_Events.Error.Error1029,FALSE,0);
Error[1030].CreateEx(TC_Events.Error.Error1030,FALSE,0);
Error[1031].CreateEx(TC_Events.Error.Error1031,FALSE,0);
Error[1032].CreateEx(TC_Events.Error.Error1032,FALSE,0);
Error[1033].CreateEx(TC_Events.Error.Error1033,FALSE,0);
Error[1034].CreateEx(TC_Events.Error.Error1034,FALSE,0);
Error[1035].CreateEx(TC_Events.Error.Error1035,FALSE,0);
Error[1036].CreateEx(TC_Events.Error.Error1036,FALSE,0);
Error[1037].CreateEx(TC_Events.Error.Error1037,FALSE,0);
Error[1038].CreateEx(TC_Events.Error.Error1038,FALSE,0);
Error[1039].CreateEx(TC_Events.Error.Error1039,FALSE,0);
Error[1040].CreateEx(TC_Events.Error.Error1040,FALSE,0);
Error[1041].CreateEx(TC_Events.Error.Error1041,FALSE,0);
Error[1042].CreateEx(TC_Events.Error.Error1042,FALSE,0);
Error[1043].CreateEx(TC_Events.Error.Error1043,FALSE,0);
Error[1044].CreateEx(TC_Events.Error.Error1044,FALSE,0);
Error[1045].CreateEx(TC_Events.Error.Error1045,FALSE,0);
Error[1046].CreateEx(TC_Events.Error.Error1046,FALSE,0);
Error[1047].CreateEx(TC_Events.Error.Error1047,FALSE,0);
Error[1048].CreateEx(TC_Events.Error.Error1048,FALSE,0);
Error[1049].CreateEx(TC_Events.Error.Error1049,FALSE,0);
Error[1050].CreateEx(TC_Events.Error.Error1050,FALSE,0);
Error[1051].CreateEx(TC_Events.Error.Error1051,FALSE,0);
Error[1052].CreateEx(TC_Events.Error.Error1052,FALSE,0);
Error[1053].CreateEx(TC_Events.Error.Error1053,FALSE,0);
Error[1054].CreateEx(TC_Events.Error.Error1054,FALSE,0);
Error[1055].CreateEx(TC_Events.Error.Error1055,FALSE,0);
Error[1056].CreateEx(TC_Events.Error.Error1056,FALSE,0);
Error[1057].CreateEx(TC_Events.Error.Error1057,FALSE,0);
Error[1058].CreateEx(TC_Events.Error.Error1058,FALSE,0);
Error[1059].CreateEx(TC_Events.Error.Error1059,FALSE,0);
Error[1060].CreateEx(TC_Events.Error.Error1060,FALSE,0);
Error[1061].CreateEx(TC_Events.Error.Error1061,FALSE,0);
Error[1062].CreateEx(TC_Events.Error.Error1062,FALSE,0);
Error[1063].CreateEx(TC_Events.Error.Error1063,FALSE,0);
Error[1064].CreateEx(TC_Events.Error.Error1064,FALSE,0);
Error[1065].CreateEx(TC_Events.Error.Error1065,FALSE,0);
Error[1066].CreateEx(TC_Events.Error.Error1066,FALSE,0);
Error[1067].CreateEx(TC_Events.Error.Error1067,FALSE,0);
Error[1068].CreateEx(TC_Events.Error.Error1068,FALSE,0);
Error[1069].CreateEx(TC_Events.Error.Error1069,FALSE,0);
Error[1070].CreateEx(TC_Events.Error.Error1070,FALSE,0);
Error[1071].CreateEx(TC_Events.Error.Error1071,FALSE,0);
Error[1072].CreateEx(TC_Events.Error.Error1072,FALSE,0);
Error[1073].CreateEx(TC_Events.Error.Error1073,FALSE,0);
Error[1074].CreateEx(TC_Events.Error.Error1074,FALSE,0);
Error[1075].CreateEx(TC_Events.Error.Error1075,FALSE,0);
Error[1076].CreateEx(TC_Events.Error.Error1076,FALSE,0);
Error[1077].CreateEx(TC_Events.Error.Error1077,FALSE,0);
Error[1078].CreateEx(TC_Events.Error.Error1078,FALSE,0);
Error[1079].CreateEx(TC_Events.Error.Error1079,FALSE,0);
Error[1080].CreateEx(TC_Events.Error.Error1080,FALSE,0);
Error[1081].CreateEx(TC_Events.Error.Error1081,FALSE,0);
Error[1082].CreateEx(TC_Events.Error.Error1082,FALSE,0);
Error[1083].CreateEx(TC_Events.Error.Error1083,FALSE,0);
Error[1084].CreateEx(TC_Events.Error.Error1084,FALSE,0);
Error[1085].CreateEx(TC_Events.Error.Error1085,FALSE,0);
Error[1086].CreateEx(TC_Events.Error.Error1086,FALSE,0);
Error[1087].CreateEx(TC_Events.Error.Error1087,FALSE,0);
Error[1088].CreateEx(TC_Events.Error.Error1088,FALSE,0);
Error[1089].CreateEx(TC_Events.Error.Error1089,FALSE,0);
Error[1090].CreateEx(TC_Events.Error.Error1090,FALSE,0);
Error[1091].CreateEx(TC_Events.Error.Error1091,FALSE,0);
Error[1092].CreateEx(TC_Events.Error.Error1092,FALSE,0);
Error[1093].CreateEx(TC_Events.Error.Error1093,FALSE,0);
Error[1094].CreateEx(TC_Events.Error.Error1094,FALSE,0);
Error[1095].CreateEx(TC_Events.Error.Error1095,FALSE,0);
Error[1096].CreateEx(TC_Events.Error.Error1096,FALSE,0);
Error[1097].CreateEx(TC_Events.Error.Error1097,FALSE,0);
Error[1098].CreateEx(TC_Events.Error.Error1098,FALSE,0);
Error[1099].CreateEx(TC_Events.Error.Error1099,FALSE,0);
Error[1100].CreateEx(TC_Events.Error.Error1100,FALSE,0);
Error[1101].CreateEx(TC_Events.Error.Error1101,FALSE,0);
Error[1102].CreateEx(TC_Events.Error.Error1102,FALSE,0);
Error[1103].CreateEx(TC_Events.Error.Error1103,FALSE,0);
Error[1104].CreateEx(TC_Events.Error.Error1104,FALSE,0);
Error[1105].CreateEx(TC_Events.Error.Error1105,FALSE,0);
Error[1106].CreateEx(TC_Events.Error.Error1106,FALSE,0);
Error[1107].CreateEx(TC_Events.Error.Error1107,FALSE,0);
Error[1108].CreateEx(TC_Events.Error.Error1108,FALSE,0);
Error[1109].CreateEx(TC_Events.Error.Error1109,FALSE,0);
Error[1110].CreateEx(TC_Events.Error.Error1110,FALSE,0);
Error[1111].CreateEx(TC_Events.Error.Error1111,FALSE,0);
Error[1112].CreateEx(TC_Events.Error.Error1112,FALSE,0);
Error[1113].CreateEx(TC_Events.Error.Error1113,FALSE,0);
Error[1114].CreateEx(TC_Events.Error.Error1114,FALSE,0);
Error[1115].CreateEx(TC_Events.Error.Error1115,FALSE,0);
Error[1116].CreateEx(TC_Events.Error.Error1116,FALSE,0);
Error[1117].CreateEx(TC_Events.Error.Error1117,FALSE,0);
Error[1118].CreateEx(TC_Events.Error.Error1118,FALSE,0);
Error[1119].CreateEx(TC_Events.Error.Error1119,FALSE,0);
Error[1120].CreateEx(TC_Events.Error.Error1120,FALSE,0);
Error[1121].CreateEx(TC_Events.Error.Error1121,FALSE,0);
Error[1122].CreateEx(TC_Events.Error.Error1122,FALSE,0);
Error[1123].CreateEx(TC_Events.Error.Error1123,FALSE,0);
Error[1124].CreateEx(TC_Events.Error.Error1124,FALSE,0);
Error[1125].CreateEx(TC_Events.Error.Error1125,FALSE,0);
Error[1126].CreateEx(TC_Events.Error.Error1126,FALSE,0);
Error[1127].CreateEx(TC_Events.Error.Error1127,FALSE,0);
Error[1128].CreateEx(TC_Events.Error.Error1128,FALSE,0);
Error[1129].CreateEx(TC_Events.Error.Error1129,FALSE,0);
Error[1130].CreateEx(TC_Events.Error.Error1130,FALSE,0);
Error[1131].CreateEx(TC_Events.Error.Error1131,FALSE,0);
Error[1132].CreateEx(TC_Events.Error.Error1132,FALSE,0);
Error[1133].CreateEx(TC_Events.Error.Error1133,FALSE,0);
Error[1134].CreateEx(TC_Events.Error.Error1134,FALSE,0);
Error[1135].CreateEx(TC_Events.Error.Error1135,FALSE,0);
Error[1136].CreateEx(TC_Events.Error.Error1136,FALSE,0);
Error[1137].CreateEx(TC_Events.Error.Error1137,FALSE,0);
Error[1138].CreateEx(TC_Events.Error.Error1138,FALSE,0);
Error[1139].CreateEx(TC_Events.Error.Error1139,FALSE,0);
Error[1140].CreateEx(TC_Events.Error.Error1140,FALSE,0);
Error[1141].CreateEx(TC_Events.Error.Error1141,FALSE,0);
Error[1142].CreateEx(TC_Events.Error.Error1142,FALSE,0);
Error[1143].CreateEx(TC_Events.Error.Error1143,FALSE,0);
Error[1144].CreateEx(TC_Events.Error.Error1144,FALSE,0);
Error[1145].CreateEx(TC_Events.Error.Error1145,FALSE,0);
Error[1146].CreateEx(TC_Events.Error.Error1146,FALSE,0);
Error[1147].CreateEx(TC_Events.Error.Error1147,FALSE,0);
Error[1148].CreateEx(TC_Events.Error.Error1148,FALSE,0);
Error[1149].CreateEx(TC_Events.Error.Error1149,FALSE,0);
Error[1150].CreateEx(TC_Events.Error.Error1150,FALSE,0);
Error[1151].CreateEx(TC_Events.Error.Error1151,FALSE,0);
Error[1152].CreateEx(TC_Events.Error.Error1152,FALSE,0);
Error[1153].CreateEx(TC_Events.Error.Error1153,FALSE,0);
Error[1154].CreateEx(TC_Events.Error.Error1154,FALSE,0);
Error[1155].CreateEx(TC_Events.Error.Error1155,FALSE,0);
Error[1156].CreateEx(TC_Events.Error.Error1156,FALSE,0);
Error[1157].CreateEx(TC_Events.Error.Error1157,FALSE,0);
Error[1158].CreateEx(TC_Events.Error.Error1158,FALSE,0);
Error[1159].CreateEx(TC_Events.Error.Error1159,FALSE,0);
Error[1160].CreateEx(TC_Events.Error.Error1160,FALSE,0);
Error[1161].CreateEx(TC_Events.Error.Error1161,FALSE,0);
Error[1162].CreateEx(TC_Events.Error.Error1162,FALSE,0);
Error[1163].CreateEx(TC_Events.Error.Error1163,FALSE,0);
